C07282=1047.858,-113.181,431.059,169.619,31.732,156.022
C07283=1047.864,-112.931,431.049,169.621,31.732,156.022
C07284=1047.869,-112.682,431.040,169.623,31.732,156.022
C07285=1047.875,-112.432,431.030,169.626,31.733,156.022
C07286=1047.881,-112.182,431.020,169.628,31.733,156.022
C07287=1047.887,-111.932,431.011,169.630,31.733,156.022
C07288=1047.894,-111.683,431.000,169.632,31.733,156.021
C07289=1047.900,-111.433,430.991,169.635,31.734,156.022
C07290=1047.906,-111.183,430.981,169.637,31.735,156.021
C07291=1047.912,-110.933,430.972,169.639,31.735,156.021
C07292=1047.918,-110.684,430.962,169.642,31.735,156.021
C07293=1047.924,-110.434,430.953,169.644,31.736,156.021
C07294=1047.931,-110.184,430.943,169.646,31.736,156.021
C07295=1047.937,-109.935,430.933,169.648,31.736,156.021
C07296=1047.942,-109.685,430.923,169.650,31.736,156.021
C07297=1047.949,-109.435,430.913,169.652,31.737,156.021
C07298=1047.955,-109.185,430.903,169.654,31.737,156.021
C07299=1047.961,-108.935,430.894,169.656,31.738,156.021
C07300=1047.967,-108.686,430.884,169.659,31.738,156.021
C07301=1047.974,-108.436,430.874,169.661,31.738,156.021
C07302=1047.980,-108.187,430.864,169.663,31.739,156.021
C07303=1047.986,-107.937,430.855,169.666,31.739,156.021
C07304=1047.992,-107.687,430.845,169.668,31.739,156.021
C07305=1047.998,-107.437,430.834,169.670,31.740,156.021
C07306=1048.005,-107.187,430.825,169.672,31.741,156.021
C07307=1048.011,-106.937,430.815,169.675,31.741,156.021
C07308=1048.017,-106.687,430.805,169.677,31.741,156.021
C07309=1048.023,-106.438,430.795,169.679,31.741,156.020
C07310=1048.029,-106.188,430.785,169.681,31.742,156.021
C07311=1048.035,-105.938,430.775,169.684,31.743,156.020
C07312=1048.042,-105.689,430.765,169.686,31.743,156.020
C07313=1048.047,-105.439,430.755,169.687,31.743,156.020
C07314=1048.053,-105.189,430.745,169.690,31.744,156.020
C07315=1048.060,-104.940,430.735,169.692,31.745,156.020
C07316=1048.066,-104.690,430.726,169.694,31.745,156.020
C07317=1048.071,-104.440,430.715,169.696,31.746,156.020
C07318=1048.078,-104.191,430.705,169.699,31.746,156.020
C07319=1048.084,-103.941,430.696,169.701,31.746,156.020
C07320=1048.090,-103.691,430.686,169.703,31.747,156.020
C07321=1048.096,-103.441,430.675,169.705,31.747,156.020
C07322=1048.103,-103.191,430.665,169.708,31.748,156.020
C07323=1048.109,-102.942,430.655,169.710,31.749,156.020
C07324=1048.114,-102.692,430.645,169.712,31.749,156.020
C07325=1048.121,-102.442,430.635,169.714,31.749,156.020
C07326=1048.127,-102.193,430.625,169.717,31.750,156.020
C07327=1048.133,-101.943,430.615,169.719,31.751,156.020
C07328=1048.139,-101.694,430.604,169.721,31.751,156.020
C07329=1048.145,-101.444,430.595,169.723,31.752,156.020
C07330=1048.152,-101.194,430.584,169.725,31.752,156.020
C07331=1048.158,-100.944,430.574,169.727,31.752,156.020
C07332=1048.164,-100.695,430.564,169.729,31.753,156.020
C07333=1048.170,-100.445,430.554,169.731,31.753,156.020
C07334=1048.176,-100.196,430.543,169.734,31.754,156.020
C07335=1048.182,-99.946,430.534,169.736,31.755,156.020
C07336=1048.189,-99.659,430.521,169.739,31.756,156.020
C07337=1048.196,-99.373,430.510,169.741,31.756,156.020
C07338=1048.203,-99.085,430.498,169.744,31.756,156.020
C07339=1048.211,-98.799,430.486,169.746,31.757,156.020
C07340=1048.220,-98.428,430.471,169.750,31.758,156.020
C07341=1048.229,-98.056,430.456,169.753,31.759,156.020
C07342=1048.238,-97.685,430.441,169.756,31.760,156.020
C07343=1048.247,-97.313,430.425,169.760,31.761,156.020
C07344=1048.254,-97.063,430.415,169.761,31.761,156.020
C07345=1048.259,-96.814,430.404,169.763,31.762,156.020
C07346=1048.266,-96.564,430.394,169.765,31.762,156.020
C07347=1048.272,-96.314,430.383,169.768,31.763,156.020
C07348=1048.278,-96.064,430.373,169.770,31.764,156.020
C07349=1048.284,-95.815,430.362,169.772,31.764,156.020
C07350=1048.290,-95.565,430.352,169.774,31.765,156.020
C07351=1048.296,-95.316,430.342,169.776,31.766,156.020
C07352=1048.302,-95.065,430.331,169.779,31.767,156.020
C07353=1048.309,-94.816,430.321,169.781,31.768,156.020
C07354=1048.314,-94.566,430.310,169.783,31.768,156.020
C07355=1048.320,-94.317,430.299,169.785,31.769,156.020
C07356=1048.326,-94.067,430.290,169.788,31.770,156.020
C07357=1048.333,-93.817,430.278,169.790,31.770,156.020
C07358=1048.339,-93.568,430.268,169.792,31.771,156.020
C07359=1048.345,-93.318,430.257,169.793,31.772,156.020
C07360=1048.350,-93.068,430.247,169.795,31.772,156.020
C07361=1048.357,-92.818,430.236,169.798,31.773,156.020
C07362=1048.363,-92.569,430.226,169.800,31.774,156.020
C07363=1048.369,-92.319,430.215,169.802,31.774,156.020
C07364=1048.375,-92.070,430.204,169.804,31.775,156.020
C07365=1048.381,-91.819,430.194,169.806,31.776,156.020
C07366=1048.388,-91.570,430.184,169.809,31.777,156.020
C07367=1048.393,-91.320,430.173,169.811,31.777,156.020
C07368=1048.400,-91.070,430.161,169.813,31.778,156.020
C07369=1048.406,-90.821,430.151,169.815,31.779,156.020
C07370=1048.412,-90.571,430.141,169.818,31.779,156.020
C07371=1048.418,-90.321,430.130,169.820,31.780,156.020
C07372=1048.425,-90.072,430.120,169.822,31.781,156.020
C07373=1048.430,-89.822,430.109,169.824,31.782,156.020
C07374=1048.437,-89.572,430.098,169.826,31.782,156.020
C07375=1048.443,-89.323,430.087,169.828,31.783,156.020
C07376=1048.449,-89.073,430.076,169.830,31.784,156.020
C07377=1048.456,-88.823,430.066,169.832,31.785,156.020
C07378=1048.461,-88.573,430.055,169.834,31.785,156.020
C07379=1048.467,-88.324,430.045,169.836,31.786,156.020
C07380=1048.474,-88.074,430.034,169.839,31.787,156.020
C07381=1048.480,-87.824,430.023,169.841,31.788,156.020
C07382=1048.486,-87.575,430.012,169.843,31.788,156.020
C07383=1048.493,-87.325,430.001,169.845,31.789,156.020
C07384=1048.498,-87.075,429.991,169.847,31.790,156.020
C07385=1048.504,-86.826,429.980,169.850,31.791,156.020
C07386=1048.511,-86.576,429.969,169.852,31.791,156.020
C07387=1048.517,-86.327,429.958,169.854,31.792,156.020
C07388=1048.523,-86.076,429.947,169.856,31.793,156.020
C07389=1048.530,-85.827,429.937,169.858,31.794,156.020
C07390=1048.536,-85.578,429.926,169.860,31.795,156.021
C07391=1048.542,-85.328,429.915,169.862,31.795,156.020
C07392=1048.548,-85.078,429.904,169.864,31.796,156.021
C07393=1048.555,-84.828,429.893,169.866,31.797,156.021
C07394=1048.560,-84.579,429.882,169.869,31.798,156.021
C07395=1048.567,-84.329,429.871,169.871,31.799,156.021
C07396=1048.577,-83.916,429.853,169.874,31.800,156.021
C07397=1048.588,-83.505,429.835,169.878,31.801,156.021
C07398=1048.598,-83.092,429.818,169.882,31.803,156.021
C07399=1048.608,-82.680,429.799,169.885,31.804,156.021
C07400=1048.615,-82.431,429.788,169.887,31.805,156.021
C07401=1048.621,-82.181,429.777,169.890,31.806,156.021
C07402=1048.627,-81.931,429.766,169.891,31.807,156.021
C07403=1048.633,-81.682,429.756,169.893,31.807,156.021
C07404=1048.640,-81.431,429.745,169.895,31.808,156.021
C07405=1048.645,-81.182,429.734,169.897,31.809,156.021
C07406=1048.652,-80.932,429.722,169.900,31.810,156.021
C07407=1048.659,-80.683,429.711,169.902,31.810,156.021
C07408=1048.665,-80.433,429.700,169.904,31.811,156.021
C07409=1048.671,-80.184,429.689,169.906,31.812,156.021
C07410=1048.677,-79.933,429.678,169.908,31.813,156.021
C07411=1048.683,-79.684,429.668,169.911,31.814,156.021
C07412=1048.690,-79.435,429.656,169.913,31.815,156.021
C07413=1048.696,-79.185,429.645,169.915,31.816,156.021
C07414=1048.702,-78.935,429.634,169.917,31.817,156.022
C07415=1048.708,-78.685,429.623,169.919,31.818,156.022
C07416=1048.715,-78.436,429.611,169.921,31.819,156.022
C07417=1048.720,-78.186,429.600,169.923,31.820,156.022
C07418=1048.727,-77.936,429.589,169.925,31.820,156.022
C07419=1048.732,-77.687,429.578,169.927,31.821,156.022
C07420=1048.739,-77.437,429.566,169.929,31.822,156.022
C07421=1048.745,-77.188,429.555,169.931,31.823,156.022
C07422=1048.751,-76.937,429.544,169.933,31.825,156.022
C07423=1048.757,-76.689,429.532,169.935,31.825,156.022
C07424=1048.764,-76.438,429.521,169.938,31.826,156.022
C07425=1048.770,-76.188,429.510,169.940,31.827,156.022
C07426=1048.776,-75.939,429.498,169.942,31.828,156.022
C07427=1048.782,-75.689,429.487,169.944,31.829,156.022
C07428=1048.788,-75.440,429.476,169.946,31.830,156.022
C07429=1048.795,-75.190,429.464,169.948,31.831,156.022
C07430=1048.800,-74.941,429.453,169.951,31.832,156.022
C07431=1048.807,-74.690,429.442,169.952,31.833,156.023
C07432=1048.813,-74.441,429.430,169.954,31.834,156.023
C07433=1048.819,-74.191,429.419,169.956,31.835,156.023
C07434=1048.826,-73.942,429.407,169.958,31.836,156.023
C07435=1048.831,-73.692,429.396,169.960,31.837,156.023
C07436=1048.838,-73.443,429.384,169.962,31.838,156.023
C07437=1048.844,-73.193,429.373,169.965,31.839,156.023
C07438=1048.849,-72.943,429.362,169.967,31.840,156.023
C07439=1048.856,-72.694,429.350,169.969,31.841,156.023
C07440=1048.862,-72.444,429.339,169.971,31.843,156.023
C07441=1048.868,-72.194,429.327,169.973,31.843,156.023
C07442=1048.874,-71.945,429.316,169.975,31.844,156.023
C07443=1048.880,-71.695,429.303,169.977,31.846,156.024
C07444=1048.886,-71.445,429.292,169.979,31.847,156.024
C07445=1048.893,-71.196,429.280,169.981,31.848,156.024
C07446=1048.898,-70.946,429.270,169.983,31.849,156.024
C07447=1048.904,-70.696,429.257,169.985,31.850,156.024
C07448=1048.911,-70.447,429.245,169.987,31.851,156.024
C07449=1048.917,-70.197,429.234,169.989,31.853,156.024
C07450=1048.923,-69.948,429.222,169.991,31.853,156.024
C07451=1048.929,-69.697,429.210,169.993,31.854,156.024
C07452=1048.935,-69.448,429.199,169.996,31.856,156.024
C07453=1048.941,-69.198,429.188,169.998,31.857,156.025
C07454=1048.947,-68.949,429.176,170.000,31.858,156.025
C07455=1048.953,-68.699,429.163,170.002,31.859,156.025
C07456=1048.959,-68.449,429.152,170.004,31.860,156.025
C07457=1048.966,-68.200,429.141,170.006,31.861,156.025
C07458=1048.971,-67.950,429.129,170.007,31.862,156.025
C07459=1048.978,-67.700,429.117,170.009,31.863,156.025
C07460=1048.984,-67.419,429.103,170.012,31.865,156.025
C07461=1048.991,-67.136,429.090,170.014,31.866,156.025
C07462=1048.999,-66.854,429.077,170.017,31.867,156.025
C07463=1049.006,-66.572,429.064,170.019,31.868,156.025
C07464=1049.011,-66.322,429.052,170.021,31.870,156.026
C07465=1049.017,-66.073,429.040,170.023,31.871,156.026
C07466=1049.024,-65.823,429.028,170.025,31.872,156.026
C07467=1049.030,-65.573,429.017,170.027,31.873,156.026
C07468=1049.036,-65.323,429.004,170.029,31.874,156.026
C07469=1049.042,-65.074,428.993,170.032,31.876,156.026
C07470=1049.049,-64.824,428.982,170.034,31.876,156.026
C07471=1049.055,-64.574,428.969,170.035,31.878,156.026
C07472=1049.061,-64.326,428.957,170.037,31.879,156.026
C07473=1049.067,-64.076,428.946,170.039,31.880,156.027
C07474=1049.073,-63.825,428.934,170.041,31.881,156.027
C07475=1049.080,-63.576,428.922,170.043,31.882,156.027
C07476=1049.086,-63.327,428.910,170.045,31.884,156.027
C07477=1049.092,-63.077,428.898,170.047,31.884,156.027
C07478=1049.098,-62.828,428.886,170.050,31.886,156.027
C07479=1049.105,-62.577,428.874,170.052,31.887,156.027
C07480=1049.110,-62.327,428.862,170.054,31.888,156.027
C07481=1049.116,-62.079,428.850,170.056,31.889,156.027
C07482=1049.123,-61.829,428.838,170.058,31.890,156.027
C07483=1049.129,-61.579,428.826,170.060,31.892,156.028
C07484=1049.135,-61.329,428.814,170.062,31.892,156.028
C07485=1049.141,-61.080,428.803,170.063,31.894,156.028
C07486=1049.147,-60.830,428.790,170.065,31.895,156.028
C07487=1049.154,-60.581,428.778,170.067,31.896,156.028
C07488=1049.161,-60.331,428.766,170.069,31.897,156.028
C07489=1049.167,-60.081,428.754,170.072,31.899,156.028
C07490=1049.173,-59.832,428.742,170.074,31.900,156.028
C07491=1049.179,-59.583,428.730,170.076,31.901,156.028
C07492=1049.185,-59.333,428.718,170.078,31.902,156.029
C07493=1049.191,-59.083,428.706,170.080,31.904,156.029
C07494=1049.198,-58.833,428.695,170.082,31.904,156.029
C07495=1049.204,-58.583,428.682,170.084,31.906,156.029
C07496=1049.211,-58.334,428.670,170.086,31.907,156.029
C07497=1049.217,-58.084,428.658,170.088,31.908,156.029
C07498=1049.223,-57.835,428.646,170.090,31.909,156.029
C07499=1049.229,-57.585,428.634,170.091,31.911,156.029
C07500=1049.235,-57.335,428.621,170.094,31.912,156.029
C07501=1049.242,-57.086,428.609,170.096,31.913,156.030
C07502=1049.248,-56.836,428.597,170.098,31.914,156.030
C07503=1049.254,-56.586,428.585,170.100,31.916,156.030
C07504=1049.261,-56.337,428.573,170.102,31.916,156.030
C07505=1049.268,-56.087,428.561,170.104,31.918,156.030
C07506=1049.274,-55.837,428.548,170.106,31.919,156.030
C07507=1049.280,-55.589,428.537,170.108,31.920,156.030
C07508=1049.286,-55.339,428.524,170.110,31.922,156.030
C07509=1049.292,-55.089,428.512,170.112,31.923,156.031
C07510=1049.299,-54.839,428.500,170.114,31.924,156.031
C07511=1049.305,-54.590,428.488,170.116,31.925,156.031
C07512=1049.311,-54.340,428.476,170.118,31.927,156.031
C07513=1049.317,-54.090,428.463,170.120,31.927,156.031
C07514=1049.324,-53.841,428.451,170.122,31.929,156.031
C07515=1049.331,-53.592,428.439,170.124,31.930,156.031
C07516=1049.337,-53.342,428.426,170.126,31.931,156.031
C07517=1049.343,-53.092,428.414,170.128,31.933,156.032
C07518=1049.349,-52.842,428.402,170.130,31.934,156.032
C07519=1049.356,-52.593,428.390,170.132,31.935,156.032
C07520=1049.362,-52.343,428.377,170.134,31.936,156.032
C07521=1049.369,-52.093,428.365,170.136,31.938,156.032
C07522=1049.375,-51.844,428.353,170.138,31.938,156.032
C07523=1049.381,-51.594,428.340,170.140,31.940,156.032
C07524=1049.389,-51.313,428.327,170.143,31.942,156.032
C07525=1049.395,-51.033,428.313,170.145,31.943,156.033
C07526=1049.403,-50.751,428.299,170.146,31.944,156.033
C07527=1049.410,-50.471,428.285,170.149,31.946,156.033
C07528=1049.416,-50.222,428.272,170.151,31.947,156.033
C07529=1049.422,-49.972,428.259,170.153,31.949,156.033
C07530=1049.429,-49.722,428.247,170.155,31.950,156.033
C07531=1049.435,-49.472,428.235,170.157,31.951,156.033
C07532=1049.441,-49.222,428.222,170.159,31.952,156.034
C07533=1049.447,-48.973,428.209,170.161,31.954,156.034
C07534=1049.454,-48.724,428.197,170.163,31.955,156.034
C07535=1049.460,-48.474,428.184,170.165,31.957,156.034
C07536=1049.466,-48.224,428.171,170.167,31.958,156.034
C07537=1049.472,-47.975,428.159,170.169,31.959,156.034
C07538=1049.478,-47.725,428.147,170.171,31.961,156.034
C07539=1049.485,-47.476,428.133,170.172,31.962,156.035
C07540=1049.490,-47.226,428.121,170.174,31.964,156.035
C07541=1049.496,-46.976,428.108,170.176,31.965,156.035
C07542=1049.503,-46.727,428.095,170.178,31.966,156.035
C07543=1049.509,-46.477,428.083,170.180,31.967,156.035
C07544=1049.515,-46.227,428.071,170.182,31.969,156.035
C07545=1049.521,-45.978,428.057,170.184,31.970,156.036
C07546=1049.527,-45.728,428.045,170.186,31.972,156.036
C07547=1049.534,-45.479,428.032,170.188,31.973,156.036
C07548=1049.540,-45.229,428.020,170.190,31.975,156.036
C07549=1049.546,-44.979,428.007,170.192,31.976,156.036
C07550=1049.552,-44.730,427.994,170.194,31.977,156.036
C07551=1049.558,-44.480,427.981,170.196,31.979,156.036
C07552=1049.565,-44.231,427.968,170.197,31.980,156.037
C07553=1049.571,-43.981,427.956,170.199,31.982,156.037
C07554=1049.577,-43.731,427.943,170.201,31.983,156.037
C07555=1049.583,-43.482,427.930,170.203,31.985,156.037
C07556=1049.590,-43.232,427.917,170.205,31.986,156.037
C07557=1049.597,-42.983,427.904,170.207,31.987,156.037
C07558=1049.603,-42.733,427.892,170.209,31.989,156.038
C07559=1049.609,-42.484,427.879,170.211,31.990,156.038
C07560=1049.615,-42.234,427.866,170.213,31.992,156.038
C07561=1049.621,-41.984,427.853,170.215,31.993,156.038
C07562=1049.627,-41.735,427.841,170.217,31.995,156.038
C07563=1049.634,-41.486,427.828,170.219,31.996,156.038
C07564=1049.640,-41.236,427.815,170.221,31.997,156.039
C07565=1049.646,-40.986,427.801,170.223,31.999,156.039
C07566=1049.652,-40.736,427.789,170.224,32.000,156.039
C07567=1049.659,-40.487,427.776,170.226,32.001,156.039
C07568=1049.666,-40.238,427.763,170.228,32.003,156.039
C07569=1049.671,-39.988,427.750,170.230,32.004,156.039
C07570=1049.678,-39.738,427.737,170.232,32.006,156.040
C07571=1049.684,-39.489,427.725,170.234,32.007,156.040
C07572=1049.690,-39.239,427.711,170.236,32.009,156.040
C07573=1049.697,-38.990,427.698,170.238,32.010,156.040
C07574=1049.703,-38.740,427.686,170.240,32.012,156.040
C07575=1049.709,-38.490,427.672,170.242,32.013,156.040
C07576=1049.715,-38.241,427.660,170.244,32.015,156.041
C07577=1049.722,-37.991,427.647,170.246,32.016,156.041
C07578=1049.728,-37.742,427.633,170.248,32.018,156.041
C07579=1049.734,-37.491,427.620,170.249,32.019,156.041
C07580=1049.740,-37.242,427.607,170.251,32.021,156.041
C07581=1049.746,-36.993,427.593,170.253,32.022,156.041
C07582=1049.752,-36.743,427.581,170.255,32.024,156.042
C07583=1049.758,-36.494,427.567,170.257,32.025,156.042
C07584=1049.764,-36.244,427.554,170.259,32.027,156.042
C07585=1049.771,-35.994,427.541,170.261,32.028,156.042
C07586=1049.777,-35.744,427.528,170.263,32.030,156.042
C07587=1049.783,-35.495,427.515,170.265,32.032,156.043
C07588=1049.790,-35.215,427.500,170.267,32.033,156.043
C07589=1049.797,-34.935,427.485,170.269,32.035,156.043
C07590=1049.804,-34.655,427.470,170.272,32.037,156.043
C07591=1049.811,-34.373,427.455,170.274,32.038,156.043
C07592=1049.817,-34.124,427.442,170.275,32.040,156.044
C07593=1049.823,-33.875,427.429,170.277,32.041,156.044
C07594=1049.830,-33.625,427.416,170.279,32.043,156.044
C07595=1049.837,-33.375,427.402,170.281,32.044,156.044
C07596=1049.842,-33.126,427.389,170.283,32.046,156.044
C07597=1049.849,-32.876,427.376,170.285,32.048,156.045
C07598=1049.855,-32.627,427.363,170.286,32.049,156.045
C07599=1049.861,-32.378,427.350,170.288,32.051,156.045
C07600=1049.867,-32.127,427.335,170.290,32.052,156.045
C07601=1049.873,-31.878,427.322,170.292,32.054,156.045
C07602=1049.879,-31.628,427.309,170.294,32.055,156.045
C07603=1049.886,-31.378,427.296,170.296,32.057,156.046
C07604=1049.892,-31.129,427.283,170.298,32.058,156.046
C07605=1049.899,-30.880,427.269,170.300,32.060,156.046
C07606=1049.905,-30.631,427.256,170.301,32.062,156.046
C07607=1049.912,-30.381,427.242,170.303,32.063,156.046
C07608=1049.918,-30.131,427.229,170.305,32.065,156.047
C07609=1049.923,-29.882,427.215,170.307,32.066,156.047
C07610=1049.930,-29.632,427.202,170.309,32.068,156.047
C07611=1049.936,-29.383,427.188,170.311,32.069,156.047
C07612=1049.942,-29.133,427.175,170.313,32.070,156.047
C07613=1049.948,-28.883,427.163,170.315,32.073,156.048
C07614=1049.955,-28.633,427.149,170.317,32.074,156.048
C07615=1049.961,-28.384,427.136,170.319,32.076,156.048
C07616=1049.968,-28.135,427.122,170.321,32.077,156.048
C07617=1049.974,-27.885,427.108,170.323,32.078,156.048
C07618=1049.980,-27.635,427.095,170.324,32.080,156.048
C07619=1049.987,-27.385,427.081,170.326,32.081,156.049
C07620=1049.993,-27.136,427.068,170.327,32.083,156.049
C07621=1049.999,-26.887,427.055,170.329,32.085,156.049
C07622=1050.006,-26.637,427.041,170.331,32.086,156.049
C07623=1050.011,-26.387,427.027,170.333,32.088,156.049
C07624=1050.018,-26.138,427.014,170.335,32.090,156.050
C07625=1050.024,-25.888,426.999,170.337,32.091,156.050
C07626=1050.030,-25.639,426.986,170.339,32.093,156.050
C07627=1050.036,-25.390,426.972,170.341,32.095,156.050
C07628=1050.043,-25.140,426.958,170.343,32.096,156.051
C07629=1050.049,-24.890,426.945,170.345,32.098,156.051
C07630=1050.055,-24.641,426.932,170.347,32.099,156.051
C07631=1050.061,-24.391,426.917,170.348,32.101,156.051
C07632=1050.067,-24.142,426.904,170.350,32.103,156.051
C07633=1050.073,-23.892,426.891,170.352,32.104,156.052
C07634=1050.080,-23.643,426.876,170.353,32.106,156.052
C07635=1050.086,-23.393,426.863,170.355,32.108,156.052
C07636=1050.092,-23.144,426.849,170.357,32.109,156.052
C07637=1050.098,-22.894,426.835,170.359,32.111,156.052
C07638=1050.105,-22.645,426.822,170.361,32.113,156.053
C07639=1050.111,-22.394,426.808,170.363,32.114,156.053
C07640=1050.117,-22.146,426.794,170.365,32.117,156.053
C07641=1050.123,-21.896,426.780,170.366,32.118,156.053
C07642=1050.129,-21.646,426.766,170.368,32.119,156.054
C07643=1050.136,-21.397,426.753,170.370,32.121,156.054
C07644=1050.142,-21.147,426.739,170.372,32.123,156.054
C07645=1050.148,-20.898,426.725,170.374,32.124,156.054
C07646=1050.154,-20.648,426.711,170.376,32.126,156.054
C07647=1050.161,-20.398,426.697,170.377,32.128,156.055
C07648=1050.167,-20.149,426.684,170.379,32.129,156.055
C07649=1050.173,-19.899,426.669,170.381,32.131,156.055
C07650=1050.179,-19.650,426.656,170.383,32.133,156.055
C07651=1050.185,-19.400,426.641,170.384,32.134,156.055
C07652=1050.193,-19.119,426.626,170.387,32.137,156.056
C07653=1050.200,-18.838,426.611,170.389,32.138,156.056
C07654=1050.207,-18.557,426.595,170.391,32.140,156.056
C07655=1050.214,-18.276,426.579,170.393,32.142,156.056
C07656=1050.219,-18.026,426.565,170.395,32.144,156.057
C07657=1050.227,-17.777,426.551,170.397,32.145,156.057
C07658=1050.233,-17.528,426.538,170.399,32.147,156.057
C07659=1050.239,-17.277,426.523,170.401,32.149,156.057
C07660=1050.245,-17.029,426.509,170.402,32.150,156.058
C07661=1050.251,-16.778,426.495,170.403,32.152,156.058
C07662=1050.258,-16.529,426.482,170.405,32.154,156.058
C07663=1050.264,-16.279,426.467,170.407,32.155,156.058
C07664=1050.270,-16.030,426.454,170.409,32.157,156.058
C07665=1050.277,-15.781,426.439,170.411,32.159,156.059
C07666=1050.283,-15.531,426.425,170.413,32.161,156.059
C07667=1050.290,-15.281,426.412,170.415,32.162,156.059
C07668=1050.296,-15.032,426.397,170.416,32.164,156.059
C07669=1050.301,-14.782,426.383,170.418,32.166,156.060
C07670=1050.309,-14.533,426.369,170.420,32.167,156.060
C07671=1050.314,-14.283,426.355,170.422,32.169,156.060
C07672=1050.320,-14.033,426.340,170.424,32.171,156.060
C07673=1050.327,-13.784,426.327,170.426,32.173,156.061
C07674=1050.333,-13.535,426.312,170.428,32.174,156.061
C07675=1050.339,-13.285,426.298,170.429,32.176,156.061
C07676=1050.346,-13.036,426.283,170.430,32.178,156.061
C07677=1050.351,-12.786,426.270,170.432,32.180,156.061
C07678=1050.358,-12.536,426.255,170.434,32.181,156.062
C07679=1050.364,-12.287,426.241,170.436,32.183,156.062
C07680=1050.370,-12.037,426.226,170.438,32.185,156.062
C07681=1050.376,-11.788,426.213,170.440,32.187,156.062
C07682=1050.383,-11.539,426.198,170.441,32.188,156.063
C07683=1050.388,-11.289,426.184,170.443,32.190,156.063
C07684=1050.395,-11.039,426.169,170.445,32.192,156.063
C07685=1050.401,-10.789,426.156,170.447,32.194,156.063
C07686=1050.407,-10.540,426.141,170.449,32.195,156.064
C07687=1050.414,-10.291,426.126,170.451,32.197,156.064
C07688=1050.420,-10.041,426.113,170.453,32.199,156.064
C07689=1050.426,-9.792,426.098,170.454,32.201,156.064
C07690=1050.432,-9.542,426.084,170.456,32.202,156.064
C07691=1050.438,-9.293,426.069,170.457,32.204,156.065
C07692=1050.445,-9.043,426.055,170.459,32.206,156.065
C07693=1050.451,-8.794,426.041,170.461,32.208,156.065
C07694=1050.457,-8.544,426.026,170.463,32.209,156.065
C07695=1050.464,-8.295,426.012,170.464,32.211,156.066
C07696=1050.470,-8.045,425.998,170.466,32.213,156.066
C07697=1050.476,-7.795,425.983,170.468,32.215,156.066
C07698=1050.482,-7.547,425.969,170.470,32.217,156.067
C07699=1050.489,-7.297,425.955,170.472,32.218,156.067
C07700=1050.495,-7.047,425.940,170.474,32.221,156.067
C07701=1050.501,-6.798,425.925,170.475,32.222,156.067
C07702=1050.508,-6.548,425.912,170.477,32.224,156.067
C07703=1050.513,-6.299,425.897,170.479,32.225,156.068
C07704=1050.520,-6.049,425.882,170.481,32.228,156.068
C07705=1050.526,-5.800,425.867,170.482,32.229,156.068
C07706=1050.532,-5.550,425.854,170.484,32.231,156.068
C07707=1050.539,-5.301,425.839,170.485,32.232,156.069
C07708=1050.545,-5.051,425.824,170.487,32.235,156.069
C07709=1050.551,-4.802,425.809,170.489,32.236,156.069
C07710=1050.558,-4.552,425.796,170.491,32.238,156.069
C07711=1050.564,-4.303,425.781,170.493,32.240,156.070
C07712=1050.570,-4.053,425.766,170.495,32.242,156.070
C07713=1050.577,-3.804,425.752,170.496,32.243,156.070
C07714=1050.583,-3.554,425.738,170.498,32.245,156.070
C07715=1050.589,-3.304,425.723,170.500,32.247,156.071
C07716=1050.596,-3.022,425.706,170.502,32.249,156.071
C07717=1050.604,-2.739,425.689,170.504,32.251,156.071
C07718=1050.610,-2.457,425.673,170.506,32.253,156.072
C07719=1050.617,-2.174,425.656,170.508,32.255,156.072
C07720=1050.622,-1.924,425.641,170.509,32.257,156.072
C07721=1050.629,-1.675,425.626,170.511,32.259,156.072
C07722=1050.635,-1.425,425.611,170.513,32.261,156.073
C07723=1050.641,-1.176,425.597,170.514,32.263,156.073
C07724=1050.647,-0.926,425.582,170.516,32.265,156.073
C07725=1050.654,-0.676,425.567,170.518,32.267,156.073
C07726=1050.659,-0.427,425.552,170.520,32.269,156.074
C07727=1050.666,-0.178,425.537,170.522,32.271,156.074
C07728=1050.672,0.072,425.523,170.523,32.272,156.074
C07729=1050.678,0.321,425.508,170.525,32.274,156.074
C07730=1050.684,0.571,425.493,170.527,32.276,156.075
C07731=1050.691,0.820,425.478,170.529,32.278,156.075
C07732=1050.697,1.070,425.463,170.531,32.280,156.075
C07733=1050.703,1.319,425.449,170.532,32.282,156.076
C07734=1050.709,1.569,425.434,170.534,32.284,156.076
C07735=1050.716,1.818,425.419,170.536,32.285,156.076
C07736=1050.722,2.068,425.404,170.537,32.287,156.076
C07737=1050.728,2.317,425.389,170.538,32.289,156.077
C07738=1050.734,2.567,425.374,170.540,32.291,156.077
C07739=1050.740,2.816,425.359,170.542,32.293,156.077
C07740=1050.746,3.065,425.344,170.544,32.295,156.077
C07741=1050.752,3.315,425.329,170.546,32.297,156.078
C07742=1050.758,3.565,425.314,170.547,32.299,156.078
C07743=1050.765,3.814,425.299,170.549,32.300,156.078
C07744=1050.771,4.064,425.284,170.551,32.302,156.078
C07745=1050.777,4.313,425.270,170.553,32.305,156.079
C07746=1050.784,4.562,425.254,170.554,32.306,156.079
C07747=1050.790,4.812,425.239,170.556,32.308,156.079
C07748=1050.796,5.061,425.224,170.558,32.310,156.080
C07749=1050.802,5.310,425.210,170.560,32.312,156.080
C07750=1050.808,5.560,425.195,170.562,32.314,156.080
C07751=1050.814,5.810,425.179,170.563,32.315,156.080
C07752=1050.820,6.060,425.164,170.564,32.318,156.081
C07753=1050.827,6.309,425.149,170.566,32.320,156.081
C07754=1050.834,6.558,425.133,170.568,32.321,156.081
C07755=1050.839,6.807,425.119,170.569,32.323,156.081
C07756=1050.846,7.057,425.104,170.571,32.325,156.082
C07757=1050.852,7.307,425.089,170.573,32.327,156.082
C07758=1050.858,7.556,425.074,170.575,32.329,156.082
C07759=1050.865,7.806,425.059,170.577,32.331,156.082
C07760=1050.871,8.055,425.043,170.578,32.333,156.083
C07761=1050.877,8.304,425.028,170.580,32.334,156.083
C07762=1050.883,8.554,425.013,170.582,32.336,156.083
C07763=1050.889,8.804,424.998,170.584,32.338,156.084
C07764=1050.896,9.053,424.983,170.585,32.340,156.084
C07765=1050.902,9.302,424.968,170.587,32.342,156.084
C07766=1050.909,9.552,424.953,170.589,32.344,156.084
C07767=1050.915,9.802,424.938,170.591,32.346,156.085
C07768=1050.921,10.051,424.922,170.592,32.348,156.085
C07769=1050.927,10.300,424.907,170.593,32.349,156.085
C07770=1050.933,10.549,424.892,170.595,32.351,156.085
C07771=1050.940,10.799,424.877,170.597,32.353,156.086
C07772=1050.946,11.048,424.862,170.599,32.355,156.086
C07773=1050.953,11.298,424.847,170.600,32.357,156.086
C07774=1050.959,11.547,424.832,170.602,32.359,156.087
C07775=1050.965,11.797,424.816,170.604,32.361,156.087
C07776=1050.971,12.046,424.800,170.606,32.362,156.087
C07777=1050.978,12.296,424.785,170.607,32.364,156.087
C07778=1050.984,12.546,424.771,170.609,32.366,156.088
C07779=1050.991,12.795,424.755,170.611,32.368,156.088
C07780=1050.998,13.079,424.738,170.613,32.371,156.088
C07781=1051.005,13.364,424.720,170.615,32.373,156.088
C07782=1051.012,13.649,424.703,170.617,32.375,156.089
C07783=1051.019,13.934,424.685,170.619,32.377,156.089
C07784=1051.026,14.183,424.670,170.621,32.379,156.089
C07785=1051.032,14.432,424.655,170.622,32.381,156.090
C07786=1051.038,14.682,424.639,170.623,32.383,156.090
C07787=1051.045,14.931,424.623,170.625,32.384,156.090
C07788=1051.051,15.181,424.608,170.627,32.386,156.090
C07789=1051.057,15.430,424.592,170.628,32.388,156.091
C07790=1051.063,15.680,424.577,170.630,32.390,156.091
C07791=1051.069,15.929,424.561,170.632,32.392,156.091
C07792=1051.076,16.179,424.546,170.634,32.394,156.092
C07793=1051.082,16.428,424.530,170.635,32.396,156.092
C07794=1051.087,16.677,424.515,170.637,32.398,156.092
C07795=1051.094,16.926,424.500,170.639,32.400,156.092
C07796=1051.100,17.176,424.484,170.640,32.402,156.093
C07797=1051.107,17.425,424.468,170.642,32.404,156.093
C07798=1051.113,17.675,424.453,170.644,32.406,156.093
C07799=1051.119,17.924,424.437,170.646,32.408,156.094
C07800=1051.125,18.174,424.422,170.647,32.410,156.094
C07801=1051.131,18.423,424.406,170.649,32.412,156.094
C07802=1051.138,18.673,424.391,170.651,32.414,156.094
C07803=1051.144,18.922,424.375,170.652,32.416,156.095
C07804=1051.150,19.172,424.360,170.653,32.418,156.095
C07805=1051.157,19.421,424.344,170.655,32.420,156.095
C07806=1051.163,19.670,424.328,170.657,32.422,156.096
C07807=1051.169,19.920,424.313,170.658,32.424,156.096
C07808=1051.175,20.169,424.297,170.660,32.426,156.096
C07809=1051.181,20.419,424.282,170.662,32.428,156.097
C07810=1051.187,20.668,424.265,170.664,32.430,156.097
C07811=1051.194,20.917,424.250,170.665,32.431,156.097
C07812=1051.200,21.167,424.234,170.667,32.433,156.097
C07813=1051.206,21.416,424.219,170.669,32.435,156.098
C07814=1051.212,21.666,424.202,170.671,32.437,156.098
C07815=1051.219,21.915,424.187,170.672,32.439,156.098
C07816=1051.225,22.165,424.171,170.674,32.441,156.099
C07817=1051.231,22.414,424.156,170.676,32.443,156.099
C07818=1051.237,22.664,424.140,170.677,32.445,156.099
C07819=1051.243,22.913,424.124,170.679,32.447,156.099
C07820=1051.250,23.163,424.108,170.681,32.449,156.100
C07821=1051.256,23.413,424.092,170.682,32.451,156.100
C07822=1051.262,23.662,424.076,170.683,32.453,156.100
C07823=1051.268,23.911,424.060,170.685,32.456,156.101
C07824=1051.275,24.160,424.045,170.687,32.458,156.101
C07825=1051.281,24.410,424.029,170.688,32.460,156.101
C07826=1051.287,24.660,424.013,170.690,32.461,156.101
C07827=1051.293,24.909,423.997,170.692,32.463,156.102
C07828=1051.299,25.158,423.981,170.693,32.465,156.102
C07829=1051.306,25.408,423.966,170.695,32.467,156.102
C07830=1051.312,25.657,423.950,170.697,32.469,156.103
C07831=1051.318,25.906,423.934,170.699,32.471,156.103
C07832=1051.324,26.155,423.918,170.700,32.473,156.103
C07833=1051.331,26.405,423.901,170.702,32.475,156.104
C07834=1051.337,26.655,423.886,170.704,32.477,156.104
C07835=1051.343,26.904,423.870,170.705,32.479,156.104
C07836=1051.350,27.153,423.854,170.707,32.481,156.105
C07837=1051.356,27.403,423.838,170.709,32.483,156.105
C07838=1051.362,27.652,423.822,170.711,32.485,156.105
C07839=1051.368,27.901,423.806,170.712,32.487,156.105
C07840=1051.374,28.151,423.791,170.714,32.489,156.106
C07841=1051.380,28.400,423.774,170.715,32.491,156.106
C07842=1051.387,28.650,423.758,170.716,32.493,156.106
C07843=1051.393,28.900,423.742,170.718,32.495,156.107
C07844=1051.400,29.185,423.724,170.720,32.497,156.107
C07845=1051.407,29.471,423.705,170.722,32.500,156.107
C07846=1051.414,29.757,423.687,170.724,32.502,156.108
C07847=1051.422,30.043,423.668,170.726,32.505,156.108
C07848=1051.428,30.292,423.652,170.727,32.507,156.108
C07849=1051.434,30.542,423.636,170.729,32.509,156.109
C07850=1051.440,30.791,423.619,170.731,32.511,156.109
C07851=1051.445,31.041,423.603,170.732,32.513,156.109
C07852=1051.453,31.290,423.587,170.734,32.515,156.110
C07853=1051.459,31.540,423.571,170.736,32.517,156.110
C07854=1051.465,31.789,423.555,170.738,32.519,156.110
C07855=1051.471,32.038,423.538,170.739,32.521,156.111
C07856=1051.477,32.288,423.522,170.741,32.523,156.111
C07857=1051.483,32.537,423.506,170.743,32.525,156.111
C07858=1051.489,32.786,423.490,170.744,32.527,156.111
C07859=1051.496,33.036,423.474,170.746,32.529,156.112
C07860=1051.502,33.285,423.457,170.748,32.531,156.112
C07861=1051.508,33.535,423.441,170.749,32.533,156.112
C07862=1051.514,33.784,423.425,170.750,32.535,156.113
C07863=1051.520,34.033,423.409,170.752,32.537,156.113
C07864=1051.527,34.283,423.392,170.753,32.539,156.113
C07865=1051.533,34.533,423.376,170.755,32.541,156.114
C07866=1051.539,34.782,423.360,170.757,32.543,156.114
C07867=1051.545,35.031,423.344,170.758,32.545,156.114
C07868=1051.551,35.280,423.328,170.760,32.547,156.114
C07869=1051.558,35.530,423.311,170.762,32.549,156.115
C07870=1051.564,35.779,423.294,170.763,32.551,156.115
C07871=1051.570,36.028,423.278,170.765,32.553,156.115
C07872=1051.576,36.278,423.262,170.767,32.555,156.116
C07873=1051.583,36.528,423.245,170.769,32.557,156.116
C07874=1051.589,36.777,423.230,170.770,32.559,156.116
C07875=1051.595,37.026,423.213,170.772,32.561,156.117
C07876=1051.601,37.276,423.197,170.774,32.563,156.117
C07877=1051.608,37.525,423.180,170.775,32.565,156.117
C07878=1051.614,37.774,423.164,170.777,32.567,156.118
C07879=1051.620,38.024,423.147,170.779,32.569,156.118
C07880=1051.626,38.273,423.131,170.780,32.572,156.118
C07881=1051.633,38.523,423.114,170.782,32.574,156.119
C07882=1051.639,38.772,423.097,170.784,32.576,156.119
C07883=1051.645,39.021,423.081,170.785,32.578,156.119
C07884=1051.651,39.270,423.065,170.786,32.580,156.120
C07885=1051.657,39.521,423.048,170.788,32.582,156.120
C07886=1051.663,39.769,423.031,170.789,32.584,156.120
C07887=1051.669,40.019,423.015,170.791,32.586,156.120
C07888=1051.675,40.268,422.999,170.793,32.588,156.121
C07889=1051.682,40.517,422.981,170.794,32.591,156.121
C07890=1051.688,40.767,422.965,170.796,32.593,156.121
C07891=1051.693,41.016,422.948,170.798,32.595,156.122
C07892=1051.699,41.266,422.932,170.799,32.597,156.122
C07893=1051.706,41.515,422.915,170.801,32.599,156.122
C07894=1051.712,41.765,422.899,170.803,32.601,156.123
C07895=1051.718,42.014,422.882,170.804,32.603,156.123
C07896=1051.725,42.263,422.865,170.806,32.605,156.123
C07897=1051.731,42.513,422.849,170.808,32.607,156.124
C07898=1051.737,42.762,422.832,170.809,32.609,156.124
C07899=1051.743,43.011,422.815,170.811,32.611,156.124
C07900=1051.750,43.261,422.799,170.813,32.613,156.125
C07901=1051.756,43.510,422.782,170.814,32.615,156.125
C07902=1051.762,43.759,422.766,170.816,32.617,156.125
C07903=1051.768,44.009,422.748,170.817,32.619,156.126
C07904=1051.774,44.258,422.731,170.819,32.622,156.126
C07905=1051.780,44.507,422.715,170.821,32.624,156.126
C07906=1051.785,44.756,422.698,170.822,32.626,156.127
C07907=1051.792,45.006,422.681,170.824,32.628,156.127
C07908=1051.799,45.292,422.661,170.825,32.631,156.127
C07909=1051.806,45.578,422.643,170.827,32.633,156.128
C07910=1051.813,45.864,422.623,170.829,32.635,156.128
C07911=1051.819,46.150,422.604,170.831,32.638,156.128
C07912=1051.826,46.399,422.587,170.832,32.640,156.129
C07913=1051.832,46.648,422.570,170.834,32.643,156.129
C07914=1051.838,46.898,422.552,170.836,32.645,156.130
C07915=1051.844,47.148,422.536,170.837,32.647,156.130
C07916=1051.850,47.396,422.519,170.839,32.649,156.130
C07917=1051.856,47.647,422.502,170.840,32.651,156.130
C07918=1051.862,47.895,422.485,170.842,32.653,156.131
C07919=1051.868,48.144,422.468,170.844,32.655,156.131
C07920=1051.875,48.394,422.451,170.845,32.657,156.131
C07921=1051.880,48.643,422.434,170.847,32.659,156.132
C07922=1051.886,48.893,422.418,170.849,32.661,156.132
C07923=1051.893,49.142,422.400,170.850,32.664,156.133
C07924=1051.898,49.392,422.383,170.852,32.666,156.133
C07925=1051.905,49.641,422.366,170.854,32.668,156.133
C07926=1051.911,49.890,422.349,170.855,32.670,156.133
C07927=1051.917,50.139,422.332,170.857,32.673,156.134
C07928=1051.924,50.389,422.315,170.859,32.675,156.134
C07929=1051.929,50.638,422.299,170.860,32.677,156.134
C07930=1051.936,50.888,422.281,170.862,32.679,156.135
C07931=1051.942,51.137,422.264,170.863,32.680,156.135
C07932=1051.947,51.386,422.247,170.865,32.683,156.136
C07933=1051.954,51.636,422.229,170.867,32.685,156.136
C07934=1051.960,51.884,422.213,170.867,32.687,156.136
C07935=1051.966,52.135,422.195,170.869,32.689,156.136
C07936=1051.972,52.384,422.178,170.871,32.691,156.137
C07937=1051.978,52.632,422.161,170.872,32.694,156.137
C07938=1051.984,52.883,422.144,170.874,32.696,156.138
C07939=1051.991,53.131,422.127,170.876,32.698,156.138
C07940=1051.997,53.381,422.110,170.877,32.700,156.138
C07941=1052.003,53.630,422.092,170.879,32.702,156.138
C07942=1052.009,53.880,422.076,170.881,32.704,156.139
C07943=1052.015,54.129,422.058,170.882,32.706,156.139
C07944=1052.022,54.378,422.041,170.884,32.708,156.139
C07945=1052.028,54.627,422.024,170.885,32.710,156.140
C07946=1052.033,54.877,422.007,170.887,32.712,156.140
C07947=1052.040,55.126,421.990,170.889,32.714,156.140
C07948=1052.046,55.375,421.973,170.890,32.717,156.141
C07949=1052.053,55.625,421.955,170.892,32.719,156.141
C07950=1052.059,55.874,421.938,170.894,32.721,156.141
C07951=1052.065,56.124,421.920,170.895,32.723,156.142
C07952=1052.071,56.372,421.904,170.897,32.725,156.142
C07953=1052.078,56.622,421.886,170.899,32.727,156.142
C07954=1052.083,56.871,421.869,170.900,32.730,156.143
C07955=1052.090,57.121,421.852,170.902,32.732,156.143
C07956=1052.095,57.370,421.834,170.904,32.734,156.143
C07957=1052.102,57.619,421.817,170.905,32.736,156.144
C07958=1052.108,57.868,421.800,170.907,32.738,156.144
C07959=1052.115,58.118,421.782,170.909,32.740,156.144
C07960=1052.121,58.367,421.765,170.910,32.742,156.145
C07961=1052.127,58.617,421.748,170.912,32.744,156.145
C07962=1052.134,58.866,421.731,170.913,32.746,156.145
C07963=1052.140,59.115,421.714,170.915,32.748,156.146
C07964=1052.146,59.365,421.696,170.916,32.750,156.146
C07965=1052.152,59.614,421.679,170.917,32.752,156.146
C07966=1052.158,59.863,421.661,170.919,32.755,156.147
C07967=1052.165,60.112,421.644,170.921,32.757,156.147
C07968=1052.171,60.362,421.627,170.922,32.759,156.147
C07969=1052.178,60.611,421.609,170.924,32.761,156.148
C07970=1052.184,60.860,421.592,170.926,32.763,156.148
C07971=1052.190,61.110,421.574,170.927,32.765,156.148
C07972=1052.197,61.396,421.554,170.929,32.767,156.149
C07973=1052.205,61.681,421.534,170.931,32.770,156.149
C07974=1052.212,61.967,421.514,170.933,32.772,156.149
C07975=1052.219,62.253,421.494,170.935,32.775,156.150
C07976=1052.225,62.501,421.477,170.937,32.777,156.150
C07977=1052.231,62.751,421.459,170.938,32.779,156.151
C07978=1052.237,63.000,421.442,170.940,32.781,156.151
C07979=1052.244,63.249,421.425,170.942,32.783,156.151
C07980=1052.250,63.499,421.407,170.943,32.785,156.151
C07981=1052.257,63.748,421.390,170.945,32.787,156.152
C07982=1052.263,63.997,421.372,170.946,32.789,156.152
C07983=1052.270,64.247,421.354,170.948,32.791,156.152
C07984=1052.275,64.496,421.337,170.950,32.793,156.153
C07985=1052.281,64.746,421.319,170.951,32.795,156.153
C07986=1052.288,64.994,421.302,170.953,32.798,156.154
C07987=1052.294,65.244,421.284,170.955,32.800,156.154
C07988=1052.300,65.494,421.266,170.956,32.802,156.154
C07989=1052.305,65.743,421.248,170.958,32.804,156.154
C07990=1052.312,65.992,421.231,170.960,32.806,156.155
C07991=1052.318,66.241,421.213,170.961,32.808,156.155
C07992=1052.324,66.490,421.195,170.963,32.810,156.156
C07993=1052.331,66.740,421.178,170.964,32.812,156.156
C07994=1052.336,66.989,421.160,170.966,32.815,156.156
C07995=1052.343,67.239,421.142,170.968,32.817,156.157
C07996=1052.349,67.488,421.125,170.969,32.819,156.157
C07997=1052.355,67.737,421.107,170.971,32.821,156.157
C07998=1052.361,67.986,421.089,170.972,32.824,156.158
C07999=1052.367,68.235,421.071,170.973,32.825,156.158
C08000=1052.374,68.485,421.054,170.975,32.827,156.158
C08001=1052.380,68.734,421.036,170.977,32.830,156.159
C08002=1052.386,68.983,421.017,170.978,32.832,156.159
C08003=1052.392,69.233,420.999,170.980,32.834,156.159
C08004=1052.399,69.482,420.982,170.981,32.836,156.160
C08005=1052.404,69.731,420.965,170.983,32.839,156.160
C08006=1052.410,69.981,420.947,170.985,32.841,156.160
C08007=1052.417,70.230,420.928,170.986,32.843,156.161
C08008=1052.422,70.479,420.910,170.988,32.845,156.161
C08009=1052.428,70.729,420.892,170.990,32.847,156.161
C08010=1052.435,70.978,420.874,170.991,32.849,156.162
C08011=1052.441,71.227,420.857,170.993,32.851,156.162
C08012=1052.447,71.476,420.839,170.995,32.854,156.162
C08013=1052.454,71.725,420.820,170.996,32.856,156.163
C08014=1052.459,71.974,420.803,170.998,32.858,156.163
C08015=1052.465,72.224,420.785,170.999,32.860,156.164
C08016=1052.472,72.473,420.766,171.001,32.862,156.164
C08017=1052.477,72.722,420.749,171.003,32.864,156.164
C08018=1052.483,72.972,420.731,171.004,32.867,156.165
C08019=1052.490,73.221,420.712,171.006,32.869,156.165
C08020=1052.496,73.471,420.694,171.008,32.871,156.165
C08021=1052.502,73.720,420.677,171.009,32.873,156.166
C08022=1052.509,73.969,420.658,171.011,32.875,156.166
C08023=1052.515,74.219,420.640,171.012,32.877,156.166
C08024=1052.521,74.467,420.622,171.014,32.879,156.167
C08025=1052.527,74.717,420.604,171.016,32.882,156.167
C08026=1052.533,74.967,420.586,171.017,32.884,156.167
C08027=1052.539,75.216,420.568,171.019,32.886,156.168
C08028=1052.545,75.465,420.550,171.021,32.889,156.168
C08029=1052.551,75.714,420.531,171.022,32.891,156.168
C08030=1052.557,75.964,420.514,171.024,32.893,156.169
C08031=1052.564,76.213,420.495,171.026,32.895,156.169
C08032=1052.569,76.462,420.477,171.027,32.897,156.169
C08033=1052.576,76.711,420.459,171.029,32.899,156.170
C08034=1052.582,76.961,420.441,171.031,32.901,156.170
C08035=1052.588,77.210,420.422,171.032,32.904,156.170
C08036=1052.595,77.495,420.401,171.034,32.906,156.171
C08037=1052.603,77.780,420.381,171.036,32.908,156.171
C08038=1052.609,78.067,420.360,171.038,32.911,156.172
C08039=1052.616,78.352,420.340,171.040,32.914,156.172
C08040=1052.623,78.601,420.321,171.041,32.915,156.172
C08041=1052.628,78.849,420.303,171.043,32.918,156.173
C08042=1052.635,79.099,420.285,171.045,32.920,156.173
C08043=1052.640,79.349,420.265,171.046,32.922,156.173
C08044=1052.646,79.598,420.248,171.047,32.925,156.174
C08045=1052.652,79.847,420.229,171.048,32.927,156.174
C08046=1052.659,80.096,420.211,171.050,32.929,156.175
C08047=1052.665,80.346,420.193,171.052,32.931,156.175
C08048=1052.670,80.595,420.173,171.053,32.933,156.175
C08049=1052.677,80.845,420.155,171.055,32.936,156.176
C08050=1052.682,81.093,420.137,171.057,32.938,156.176
C08051=1052.689,81.342,420.119,171.058,32.940,156.176
C08052=1052.695,81.592,420.101,171.060,32.942,156.177
C08053=1052.701,81.841,420.082,171.061,32.944,156.177
C08054=1052.706,82.090,420.063,171.063,32.947,156.177
C08055=1052.713,82.340,420.045,171.065,32.949,156.178
C08056=1052.719,82.589,420.027,171.066,32.951,156.178
C08057=1052.725,82.838,420.008,171.068,32.953,156.179
C08058=1052.732,83.087,419.989,171.070,32.955,156.179
C08059=1052.737,83.337,419.971,171.071,32.957,156.179
C08060=1052.743,83.585,419.952,171.073,32.960,156.180
C08061=1052.749,83.835,419.934,171.075,32.962,156.180
C08062=1052.756,84.084,419.916,171.076,32.964,156.180
C08063=1052.762,84.333,419.897,171.078,32.966,156.181
C08064=1052.768,84.583,419.878,171.079,32.968,156.181
C08065=1052.774,84.832,419.859,171.081,32.971,156.181
C08066=1052.780,85.081,419.842,171.083,32.973,156.182
C08067=1052.786,85.330,419.823,171.084,32.975,156.182
C08068=1052.792,85.580,419.804,171.086,32.978,156.182
C08069=1052.798,85.829,419.785,171.088,32.980,156.183
C08070=1052.805,86.078,419.767,171.089,32.982,156.183
C08071=1052.811,86.328,419.749,171.091,32.984,156.184
C08072=1052.817,86.577,419.730,171.093,32.986,156.184
C08073=1052.823,86.826,419.711,171.094,32.988,156.184
C08074=1052.829,87.075,419.692,171.096,32.991,156.185
C08075=1052.835,87.324,419.674,171.098,32.993,156.185
C08076=1052.842,87.573,419.655,171.099,32.995,156.185
C08077=1052.847,87.823,419.637,171.101,32.997,156.186
C08078=1052.853,88.072,419.618,171.103,32.999,156.186
C08079=1052.860,88.321,419.599,171.104,33.001,156.186
C08080=1052.866,88.570,419.581,171.106,33.004,156.187
C08081=1052.872,88.820,419.561,171.107,33.006,156.187
C08082=1052.878,89.069,419.543,171.109,33.008,156.187
C08083=1052.885,89.318,419.524,171.111,33.010,156.188
C08084=1052.891,89.567,419.505,171.112,33.012,156.188
C08085=1052.897,89.817,419.487,171.114,33.014,156.188
C08086=1052.903,90.066,419.468,171.116,33.016,156.189
C08087=1052.909,90.315,419.450,171.117,33.019,156.189
C08088=1052.916,90.564,419.431,171.119,33.021,156.189
C08089=1052.921,90.813,419.412,171.121,33.023,156.190
C08090=1052.927,91.062,419.393,171.122,33.025,156.190
C08091=1052.933,91.312,419.374,171.124,33.027,156.191
C08092=1052.939,91.561,419.356,171.126,33.030,156.191
C08093=1052.945,91.810,419.336,171.127,33.032,156.191
C08094=1052.952,92.059,419.318,171.129,33.034,156.192
C08095=1052.957,92.309,419.298,171.131,33.036,156.192
C08096=1052.964,92.558,419.280,171.132,33.039,156.192
C08097=1052.969,92.807,419.261,171.134,33.041,156.193
C08098=1052.976,93.057,419.242,171.136,33.044,156.193
C08099=1052.981,93.306,419.223,171.137,33.045,156.194
C08100=1052.988,93.591,419.201,171.139,33.048,156.194
C08101=1052.995,93.876,419.179,171.141,33.051,156.194
C08102=1053.002,94.162,419.157,171.143,33.053,156.195
C08103=1053.009,94.447,419.135,171.145,33.056,156.195
C08104=1053.016,94.696,419.116,171.146,33.058,156.196
C08105=1053.021,94.946,419.097,171.148,33.060,156.196
C08106=1053.028,95.195,419.079,171.150,33.062,156.196
C08107=1053.033,95.444,419.059,171.151,33.064,156.197
C08108=1053.040,95.693,419.041,171.153,33.067,156.197
C08109=1053.046,95.942,419.021,171.155,33.069,156.197
C08110=1053.052,96.191,419.002,171.156,33.072,156.198
C08111=1053.058,96.441,418.983,171.158,33.074,156.198
C08112=1053.064,96.690,418.964,171.160,33.076,156.198
C08113=1053.070,96.939,418.945,171.161,33.078,156.199
C08114=1053.076,97.189,418.926,171.163,33.080,156.199
C08115=1053.082,97.437,418.906,171.165,33.083,156.200
C08116=1053.088,97.687,418.887,171.166,33.085,156.200
C08117=1053.095,97.936,418.868,171.168,33.087,156.200
C08118=1053.100,98.185,418.849,171.170,33.089,156.201
C08119=1053.107,98.434,418.831,171.171,33.091,156.201
C08120=1053.113,98.683,418.811,171.173,33.093,156.201
C08121=1053.119,98.932,418.792,171.175,33.096,156.202
C08122=1053.125,99.182,418.773,171.176,33.098,156.202
C08123=1053.130,99.431,418.753,171.178,33.100,156.203
C08124=1053.137,99.680,418.734,171.180,33.102,156.203
C08125=1053.143,99.929,418.715,171.181,33.104,156.203
C08126=1053.149,100.178,418.696,171.183,33.107,156.204
C08127=1053.156,100.428,418.677,171.185,33.109,156.204
C08128=1053.162,100.677,418.657,171.186,33.111,156.204
C08129=1053.168,100.926,418.638,171.188,33.113,156.205
C08130=1053.174,101.176,418.619,171.190,33.115,156.205
C08131=1053.180,101.425,418.599,171.191,33.118,156.205
C08132=1053.186,101.674,418.580,171.193,33.120,156.206
C08133=1053.192,101.923,418.561,171.195,33.122,156.206
C08134=1053.198,102.172,418.541,171.196,33.124,156.206
C08135=1053.203,102.421,418.522,171.198,33.127,156.207
C08136=1053.209,102.670,418.502,171.200,33.129,156.207
C08137=1053.216,102.919,418.483,171.201,33.131,156.208
C08138=1053.222,103.169,418.464,171.203,33.133,156.208
C08139=1053.228,103.418,418.444,171.205,33.136,156.208
C08140=1053.233,103.667,418.425,171.206,33.138,156.209
C08141=1053.239,103.916,418.405,171.208,33.140,156.209
C08142=1053.246,104.166,418.386,171.210,33.142,156.209
C08143=1053.252,104.415,418.366,171.211,33.145,156.210
C08144=1053.258,104.664,418.346,171.213,33.147,156.210
C08145=1053.264,104.913,418.327,171.215,33.150,156.211
C08146=1053.270,105.162,418.307,171.216,33.152,156.211
C08147=1053.275,105.412,418.288,171.218,33.154,156.211
C08148=1053.282,105.660,418.269,171.220,33.156,156.212
C08149=1053.288,105.910,418.249,171.221,33.159,156.212
C08150=1053.294,106.158,418.229,171.223,33.161,156.212
C08151=1053.300,106.408,418.210,171.225,33.163,156.213
C08152=1053.306,106.657,418.190,171.226,33.165,156.213
C08153=1053.312,106.906,418.171,171.228,33.167,156.214
C08154=1053.318,107.155,418.151,171.230,33.170,156.214
C08155=1053.324,107.405,418.132,171.231,33.172,156.214
C08156=1053.330,107.653,418.112,171.233,33.174,156.215
C08157=1053.336,107.903,418.093,171.235,33.176,156.215
C08158=1053.342,108.152,418.072,171.237,33.179,156.215
C08159=1053.348,108.401,418.053,171.238,33.181,156.216
C08160=1053.355,108.650,418.034,171.240,33.183,156.216
C08161=1053.361,108.899,418.014,171.242,33.185,156.217
C08162=1053.367,109.149,417.995,171.243,33.187,156.217
C08163=1053.373,109.398,417.974,171.245,33.190,156.217
C08164=1053.380,109.683,417.952,171.247,33.192,156.218
C08165=1053.387,109.969,417.929,171.249,33.195,156.218
C08166=1053.393,110.254,417.907,171.251,33.198,156.219
C08167=1053.401,110.539,417.884,171.253,33.200,156.219
C08168=1053.407,110.789,417.865,171.254,33.202,156.219
C08169=1053.413,111.037,417.845,171.256,33.204,156.220
C08170=1053.420,111.287,417.825,171.258,33.207,156.220
C08171=1053.425,111.536,417.806,171.260,33.209,156.220
C08172=1053.431,111.785,417.786,171.261,33.211,156.221
C08173=1053.437,112.034,417.766,171.263,33.213,156.221
C08174=1053.443,112.284,417.746,171.265,33.216,156.222
C08175=1053.449,112.533,417.726,171.266,33.218,156.222
C08176=1053.455,112.782,417.706,171.268,33.220,156.222
C08177=1053.461,113.031,417.686,171.270,33.222,156.223
C08178=1053.467,113.280,417.667,171.271,33.225,156.223
C08179=1053.474,113.530,417.647,171.273,33.227,156.223
C08180=1053.480,113.778,417.627,171.275,33.229,156.224
C08181=1053.486,114.027,417.607,171.277,33.231,156.224
C08182=1053.491,114.277,417.587,171.278,33.234,156.225
C08183=1053.497,114.526,417.567,171.280,33.236,156.225
C08184=1053.503,114.775,417.547,171.282,33.238,156.225
C08185=1053.509,115.024,417.527,171.283,33.241,156.226
C08186=1053.515,115.273,417.507,171.285,33.243,156.226
C08187=1053.521,115.522,417.486,171.287,33.246,156.227
C08188=1053.527,115.771,417.466,171.288,33.248,156.227
C08189=1053.533,116.021,417.447,171.290,33.250,156.227
C08190=1053.539,116.270,417.427,171.292,33.253,156.228
C08191=1053.544,116.519,417.406,171.293,33.255,156.228
C08192=1053.550,116.768,417.386,171.295,33.257,156.229
C08193=1053.557,117.017,417.366,171.297,33.260,156.229
C08194=1053.563,117.266,417.346,171.299,33.262,156.229
C08195=1053.568,117.515,417.325,171.300,33.264,156.230
C08196=1053.574,117.764,417.305,171.302,33.266,156.230
C08197=1053.580,118.013,417.285,171.304,33.269,156.230
C08198=1053.586,118.263,417.264,171.305,33.271,156.231
C08199=1053.592,118.511,417.244,171.307,33.273,156.231
C08200=1053.598,118.760,417.224,171.309,33.276,156.232
C08201=1053.604,119.010,417.205,171.311,33.278,156.232
C08202=1053.609,119.259,417.184,171.312,33.280,156.232
C08203=1053.615,119.508,417.164,171.314,33.282,156.233
C08204=1053.622,119.758,417.144,171.316,33.285,156.233
C08205=1053.628,120.007,417.124,171.317,33.287,156.234
C08206=1053.633,120.256,417.104,171.319,33.289,156.234
C08207=1053.639,120.505,417.084,171.321,33.292,156.234
C08208=1053.646,120.754,417.063,171.323,33.294,156.235
C08209=1053.651,121.003,417.042,171.324,33.296,156.235
C08210=1053.657,121.251,417.022,171.326,33.298,156.235
C08211=1053.664,121.501,417.002,171.328,33.301,156.236
C08212=1053.669,121.750,416.981,171.329,33.303,156.236
C08213=1053.675,121.999,416.961,171.331,33.306,156.237
C08214=1053.682,122.248,416.941,171.333,33.308,156.237
C08215=1053.688,122.497,416.921,171.335,33.310,156.237
C08216=1053.693,122.746,416.900,171.336,33.313,156.238
C08217=1053.700,122.996,416.880,171.338,33.315,156.238
C08218=1053.706,123.245,416.860,171.340,33.317,156.239
C08219=1053.711,123.494,416.839,171.342,33.319,156.239
C08220=1053.717,123.743,416.819,171.343,33.322,156.239
C08221=1053.724,123.991,416.798,171.345,33.324,156.240
C08222=1053.730,124.241,416.778,171.347,33.326,156.240
C08223=1053.736,124.490,416.758,171.349,33.328,156.240
C08224=1053.742,124.739,416.738,171.350,33.331,156.241
C08225=1053.747,124.989,416.717,171.352,33.333,156.241
C08226=1053.753,125.238,416.697,171.354,33.335,156.242
C08227=1053.760,125.486,416.676,171.356,33.338,156.242
C08228=1053.766,125.772,416.653,171.358,33.340,156.243
C08229=1053.773,126.057,416.630,171.360,33.343,156.243
C08230=1053.780,126.343,416.606,171.362,33.346,156.243
C08231=1053.787,126.628,416.582,171.364,33.348,156.244
C08232=1053.793,126.877,416.562,171.365,33.350,156.244
C08233=1053.799,127.127,416.541,171.367,33.353,156.245
C08234=1053.806,127.375,416.521,171.369,33.355,156.245
C08235=1053.812,127.624,416.500,171.371,33.357,156.245
C08236=1053.817,127.873,416.480,171.372,33.359,156.246
C08237=1053.824,128.122,416.459,171.374,33.362,156.246
C08238=1053.830,128.371,416.439,171.376,33.364,156.246
C08239=1053.836,128.621,416.418,171.378,33.366,156.247
C08240=1053.842,128.870,416.398,171.379,33.368,156.247
C08241=1053.849,129.119,416.377,171.381,33.371,156.248
C08242=1053.854,129.368,416.356,171.383,33.373,156.248
C08243=1053.861,129.617,416.336,171.385,33.375,156.248
C08244=1053.867,129.865,416.315,171.388,33.378,156.249
C08245=1053.873,130.115,416.294,171.389,33.380,156.249
C08246=1053.879,130.364,416.274,171.391,33.382,156.250
C08247=1053.885,130.613,416.253,171.393,33.384,156.250
C08248=1053.891,130.862,416.233,171.395,33.387,156.250
C08249=1053.898,131.112,416.213,171.396,33.389,156.251
C08250=1053.903,131.360,416.191,171.398,33.391,156.251
C08251=1053.910,131.610,416.171,171.400,33.393,156.251
C08252=1053.916,131.858,416.150,171.402,33.396,156.252
C08253=1053.922,132.108,416.129,171.404,33.398,156.252
C08254=1053.928,132.356,416.108,171.405,33.400,156.253
C08255=1053.934,132.606,416.087,171.407,33.403,156.253
C08256=1053.940,132.855,416.067,171.409,33.405,156.253
C08257=1053.945,133.103,416.046,171.411,33.408,156.254
C08258=1053.951,133.353,416.025,171.412,33.410,156.254
C08259=1053.957,133.601,416.004,171.414,33.412,156.255
C08260=1053.963,133.851,415.983,171.416,33.415,156.255
C08261=1053.969,134.100,415.962,171.418,33.417,156.255
C08262=1053.975,134.349,415.942,171.420,33.419,156.256
C08263=1053.981,134.598,415.921,171.421,33.422,156.256
C08264=1053.987,134.847,415.899,171.423,33.424,156.257
C08265=1053.994,135.096,415.879,171.425,33.426,156.257
C08266=1053.999,135.345,415.857,171.427,33.429,156.257
C08267=1054.005,135.595,415.836,171.429,33.431,156.258
C08268=1054.011,135.843,415.816,171.430,33.433,156.258
C08269=1054.017,136.093,415.795,171.432,33.436,156.259
C08270=1054.023,136.341,415.774,171.434,33.438,156.259
C08271=1054.030,136.590,415.752,171.436,33.440,156.259
C08272=1054.035,136.839,415.732,171.437,33.442,156.260
C08273=1054.041,137.088,415.710,171.439,33.445,156.260
C08274=1054.047,137.337,415.690,171.441,33.447,156.261
C08275=1054.053,137.586,415.669,171.443,33.449,156.261
C08276=1054.059,137.836,415.647,171.445,33.452,156.261
C08277=1054.065,138.085,415.626,171.447,33.454,156.262
C08278=1054.071,138.334,415.605,171.448,33.456,156.262
C08279=1054.077,138.582,415.584,171.450,33.459,156.263
C08280=1054.083,138.832,415.563,171.452,33.461,156.263
C08281=1054.089,139.081,415.542,171.454,33.463,156.263
C08282=1054.095,139.329,415.521,171.456,33.466,156.264
C08283=1054.101,139.579,415.500,171.457,33.468,156.264
C08284=1054.107,139.828,415.479,171.459,33.470,156.264
C08285=1054.113,140.077,415.457,171.461,33.473,156.265
C08286=1054.119,140.326,415.435,171.463,33.476,156.265
C08287=1054.125,140.575,415.416,171.465,33.478,156.266
C08288=1054.131,140.824,415.394,171.467,33.480,156.266
C08289=1054.137,141.073,415.373,171.469,33.483,156.267
C08290=1054.143,141.322,415.351,171.471,33.485,156.267
C08291=1054.149,141.570,415.330,171.473,33.487,156.267
C08292=1054.155,141.856,415.305,171.475,33.490,156.268
C08293=1054.162,142.141,415.281,171.477,33.493,156.268
C08294=1054.168,142.427,415.257,171.479,33.495,156.269
C08295=1054.176,142.711,415.232,171.481,33.498,156.269
C08296=1054.182,142.961,415.211,171.483,33.501,156.270
C08297=1054.188,143.210,415.189,171.485,33.503,156.270
C08298=1054.194,143.458,415.168,171.487,33.505,156.270
C08299=1054.200,143.707,415.146,171.489,33.508,156.271
C08300=1054.206,143.957,415.125,171.490,33.510,156.271
C08301=1054.211,144.206,415.104,171.492,33.512,156.272
C08302=1054.217,144.455,415.082,171.494,33.515,156.272
C08303=1054.224,144.704,415.061,171.496,33.517,156.272
C08304=1054.229,144.953,415.040,171.498,33.520,156.273
C08305=1054.236,145.202,415.019,171.500,33.522,156.273
C08306=1054.242,145.451,414.997,171.501,33.524,156.274
C08307=1054.248,145.699,414.976,171.503,33.527,156.274
C08308=1054.254,145.949,414.954,171.505,33.529,156.274
C08309=1054.260,146.198,414.932,171.507,33.531,156.275
C08310=1054.266,146.447,414.911,171.509,33.534,156.275
C08311=1054.272,146.695,414.889,171.511,33.536,156.276
C08312=1054.278,146.945,414.868,171.513,33.538,156.276
C08313=1054.284,147.194,414.846,171.514,33.541,156.277
C08314=1054.290,147.442,414.825,171.516,33.543,156.277
C08315=1054.296,147.692,414.803,171.518,33.546,156.277
C08316=1054.302,147.941,414.782,171.520,33.548,156.278
C08317=1054.308,148.190,414.760,171.522,33.551,156.278
C08318=1054.314,148.438,414.739,171.524,33.553,156.279
C08319=1054.320,148.688,414.717,171.526,33.555,156.279
C08320=1054.325,148.937,414.695,171.528,33.558,156.279
C08321=1054.331,149.186,414.674,171.530,33.560,156.280
C08322=1054.337,149.435,414.652,171.532,33.563,156.280
C08323=1054.343,149.684,414.630,171.534,33.565,156.281
C08324=1054.349,149.933,414.609,171.536,33.567,156.281
C08325=1054.355,150.181,414.587,171.538,33.570,156.281
C08326=1054.361,150.430,414.565,171.540,33.572,156.282
C08327=1054.368,150.680,414.543,171.541,33.574,156.282
C08328=1054.373,150.929,414.521,171.543,33.577,156.283
C08329=1054.379,151.178,414.500,171.545,33.579,156.283
C08330=1054.385,151.427,414.478,171.547,33.582,156.284
C08331=1054.391,151.675,414.456,171.549,33.585,156.284
C08332=1054.397,151.925,414.434,171.551,33.586,156.284
C08333=1054.402,152.173,414.412,171.553,33.589,156.285
C08334=1054.408,152.423,414.391,171.555,33.592,156.285
C08335=1054.414,152.672,414.369,171.556,33.594,156.286
C08336=1054.421,152.920,414.347,171.558,33.597,156.286
C08337=1054.427,153.169,414.326,171.560,33.599,156.286
C08338=1054.432,153.418,414.303,171.562,33.601,156.287
C08339=1054.438,153.668,414.282,171.564,33.604,156.287
C08340=1054.445,153.916,414.259,171.566,33.606,156.288
C08341=1054.451,154.165,414.238,171.568,33.609,156.288
C08342=1054.456,154.414,414.216,171.570,33.611,156.289
C08343=1054.462,154.663,414.194,171.572,33.613,156.289
C08344=1054.468,154.912,414.172,171.574,33.616,156.289
C08345=1054.474,155.161,414.150,171.575,33.618,156.290
C08346=1054.480,155.410,414.127,171.578,33.621,156.290
C08347=1054.486,155.659,414.106,171.580,33.623,156.291
C08348=1054.492,155.908,414.084,171.582,33.625,156.291
C08349=1054.498,156.157,414.061,171.584,33.628,156.291
C08350=1054.504,156.406,414.040,171.586,33.631,156.292
C08351=1054.510,156.655,414.018,171.588,33.633,156.292
C08352=1054.516,156.904,413.995,171.590,33.636,156.293
C08353=1054.522,157.153,413.974,171.592,33.638,156.293
C08354=1054.528,157.401,413.952,171.594,33.640,156.294
C08355=1054.533,157.651,413.929,171.596,33.643,156.294
C08356=1054.540,157.935,413.904,171.598,33.646,156.295
C08357=1054.546,158.220,413.879,171.600,33.648,156.295
C08358=1054.554,158.506,413.853,171.602,33.652,156.296
C08359=1054.561,158.790,413.828,171.604,33.654,156.296
C08360=1054.567,159.040,413.806,171.606,33.657,156.296
C08361=1054.573,159.288,413.784,171.608,33.659,156.297
C08362=1054.578,159.537,413.762,171.610,33.661,156.297
C08363=1054.584,159.786,413.740,171.612,33.664,156.298
C08364=1054.591,160.035,413.718,171.614,33.666,156.298
C08365=1054.596,160.284,413.695,171.616,33.669,156.299
C08366=1054.603,160.533,413.673,171.618,33.671,156.299
C08367=1054.608,160.782,413.650,171.620,33.674,156.299
C08368=1054.615,161.030,413.628,171.622,33.676,156.300
C08369=1054.620,161.280,413.606,171.625,33.679,156.300
C08370=1054.626,161.529,413.583,171.627,33.682,156.301
C08371=1054.631,161.777,413.562,171.628,33.684,156.301
C08372=1054.637,162.026,413.539,171.630,33.687,156.302
C08373=1054.643,162.275,413.516,171.632,33.689,156.302
C08374=1054.648,162.525,413.493,171.634,33.692,156.303
C08375=1054.655,162.773,413.471,171.636,33.694,156.303
C08376=1054.661,163.022,413.448,171.638,33.697,156.303
C08377=1054.666,163.272,413.426,171.640,33.699,156.304
C08378=1054.671,163.520,413.403,171.642,33.702,156.304
C08379=1054.678,163.768,413.381,171.644,33.704,156.305
C08380=1054.683,164.017,413.358,171.646,33.707,156.305
C08381=1054.689,164.267,413.336,171.648,33.710,156.306
C08382=1054.694,164.516,413.313,171.650,33.712,156.306
C08383=1054.701,164.764,413.291,171.652,33.715,156.307
C08384=1054.707,165.013,413.268,171.654,33.717,156.307
C08385=1054.712,165.263,413.245,171.656,33.720,156.308
C08386=1054.718,165.512,413.222,171.658,33.723,156.308
C08387=1054.724,165.760,413.200,171.660,33.725,156.308
C08388=1054.730,166.009,413.177,171.662,33.728,156.309
C08389=1054.735,166.257,413.155,171.664,33.730,156.309
C08390=1054.741,166.507,413.132,171.666,33.733,156.310
C08391=1054.747,166.755,413.110,171.668,33.735,156.310
C08392=1054.753,167.004,413.087,171.670,33.738,156.311
C08393=1054.758,167.253,413.064,171.672,33.741,156.311
C08394=1054.764,167.502,413.041,171.674,33.743,156.312
C08395=1054.770,167.751,413.018,171.676,33.746,156.312
C08396=1054.776,168.000,412.997,171.678,33.748,156.312
C08397=1054.782,168.249,412.974,171.680,33.751,156.313
C08398=1054.788,168.498,412.951,171.682,33.753,156.313
C08399=1054.793,168.747,412.928,171.684,33.756,156.314
C08400=1054.799,168.996,412.905,171.686,33.758,156.314
C08401=1054.806,169.244,412.882,171.688,33.761,156.315
C08402=1054.811,169.493,412.859,171.690,33.763,156.315
C08403=1054.817,169.742,412.836,171.692,33.766,156.316
C08404=1054.823,169.991,412.814,171.694,33.769,156.316
C08405=1054.828,170.240,412.791,171.696,33.771,156.316
C08406=1054.835,170.489,412.768,171.699,33.774,156.317
C08407=1054.841,170.737,412.745,171.701,33.777,156.317
C08408=1054.846,170.986,412.722,171.703,33.779,156.318
C08409=1054.853,171.236,412.699,171.705,33.782,156.318
C08410=1054.858,171.485,412.676,171.707,33.784,156.319
C08411=1054.865,171.733,412.654,171.709,33.787,156.319
C08412=1054.871,171.982,412.631,171.711,33.789,156.320
C08413=1054.876,172.231,412.608,171.713,33.792,156.320
C08414=1054.882,172.480,412.585,171.715,33.795,156.321
C08415=1054.888,172.729,412.562,171.717,33.797,156.321
C08416=1054.894,172.978,412.539,171.719,33.800,156.321
C08417=1054.900,173.226,412.517,171.721,33.802,156.322
C08418=1054.906,173.475,412.494,171.723,33.805,156.322
C08419=1054.911,173.724,412.471,171.725,33.807,156.323
C08420=1054.919,174.009,412.444,171.728,33.810,156.323
C08421=1054.925,174.294,412.418,171.730,33.813,156.324
C08422=1054.932,174.578,412.392,171.732,33.816,156.324
C08423=1054.939,174.862,412.365,171.736,33.819,156.325
C08424=1054.944,175.111,412.342,171.738,33.822,156.325
C08425=1054.951,175.360,412.320,171.740,33.824,156.326
C08426=1054.957,175.609,412.297,171.742,33.827,156.326
C08427=1054.963,175.858,412.273,171.744,33.829,156.327
C08428=1054.969,176.106,412.250,171.746,33.832,156.327
C08429=1054.975,176.355,412.227,171.748,33.834,156.328
C08430=1054.981,176.604,412.204,171.750,33.837,156.328
C08431=1054.986,176.853,412.181,171.752,33.840,156.328
C08432=1054.994,177.102,412.158,171.754,33.842,156.329
C08433=1054.999,177.351,412.135,171.756,33.845,156.329
C08434=1055.005,177.600,412.112,171.758,33.847,156.330
C08435=1055.011,177.848,412.089,171.760,33.850,156.330
C08436=1055.017,178.097,412.065,171.762,33.853,156.331
C08437=1055.023,178.346,412.042,171.765,33.855,156.331
C08438=1055.029,178.595,412.019,171.768,33.858,156.332
C08439=1055.035,178.844,411.996,171.770,33.860,156.332
C08440=1055.042,179.123,411.970,171.772,33.863,156.333
C08441=1055.049,179.401,411.944,171.774,33.866,156.333
C08442=1055.055,179.680,411.918,171.777,33.869,156.334
C08443=1055.062,179.958,411.892,171.779,33.872,156.334
C08444=1055.068,180.207,411.869,171.781,33.874,156.335
C08445=1055.074,180.455,411.845,171.783,33.877,156.335
C08446=1055.080,180.704,411.822,171.785,33.879,156.336
C08447=1055.086,180.953,411.799,171.787,33.882,156.336
C08448=1055.093,181.202,411.775,171.790,33.885,156.336
C08449=1055.098,181.451,411.752,171.792,33.887,156.337
C08450=1055.104,181.699,411.729,171.794,33.890,156.337
C08451=1055.111,181.949,411.706,171.796,33.893,156.338
C08452=1055.117,182.197,411.682,171.798,33.895,156.338
C08453=1055.123,182.446,411.659,171.801,33.898,156.339
C08454=1055.130,182.695,411.635,171.803,33.900,156.339
C08455=1055.136,182.944,411.612,171.805,33.903,156.340
C08456=1055.141,183.193,411.589,171.808,33.905,156.340
C08457=1055.148,183.442,411.565,171.810,33.908,156.341
C08458=1055.154,183.691,411.542,171.812,33.911,156.341
C08459=1055.160,183.939,411.519,171.814,33.913,156.341
C08460=1055.166,184.188,411.495,171.816,33.916,156.342
C08461=1055.172,184.437,411.472,171.818,33.919,156.342
C08462=1055.177,184.685,411.447,171.820,33.921,156.343
C08463=1055.184,184.935,411.424,171.822,33.924,156.343
C08464=1055.190,185.183,411.401,171.824,33.927,156.344
C08465=1055.195,185.432,411.377,171.827,33.929,156.344
C08466=1055.201,185.681,411.353,171.830,33.933,156.345
C08467=1055.207,185.930,411.329,171.832,33.935,156.345
C08468=1055.212,186.179,411.306,171.834,33.938,156.346
C08469=1055.218,186.427,411.281,171.836,33.941,156.346
C08470=1055.224,186.676,411.258,171.838,33.943,156.347
C08471=1055.230,186.925,411.234,171.840,33.946,156.347
C08472=1055.235,187.174,411.210,171.842,33.949,156.348
C08473=1055.241,187.422,411.187,171.845,33.951,156.348
C08474=1055.247,187.671,411.162,171.847,33.955,156.349
C08475=1055.253,187.920,411.139,171.849,33.957,156.349
C08476=1055.258,188.169,411.115,171.851,33.960,156.350
C08477=1055.265,188.418,411.091,171.853,33.963,156.350
C08478=1055.270,188.667,411.066,171.855,33.965,156.351
C08479=1055.276,188.915,411.043,171.858,33.968,156.351
C08480=1055.282,189.165,411.019,171.860,33.971,156.352
C08481=1055.288,189.413,410.995,171.863,33.973,156.352
C08482=1055.294,189.661,410.972,171.865,33.977,156.353
C08483=1055.300,189.911,410.947,171.867,33.979,156.353
C08484=1055.306,190.164,410.923,171.869,33.982,156.354
C08485=1055.311,190.419,410.898,171.871,33.985,156.354
C08486=1055.318,190.674,410.874,171.874,33.988,156.355
C08487=1055.323,190.928,410.849,171.876,33.990,156.355
C08488=1055.330,191.177,410.825,171.878,33.994,156.356
C08489=1055.335,191.425,410.801,171.880,33.996,156.356
C08490=1055.341,191.674,410.777,171.883,33.999,156.357
C08491=1055.347,191.923,410.753,171.885,34.002,156.357
C08492=1055.353,192.172,410.730,171.888,34.004,156.358
C08493=1055.359,192.421,410.705,171.890,34.007,156.358
C08494=1055.365,192.669,410.681,171.892,34.010,156.359
C08495=1055.371,192.919,410.657,171.894,34.013,156.359
C08496=1055.377,193.167,410.633,171.896,34.016,156.360
C08497=1055.382,193.415,410.609,171.899,34.019,156.360
C08498=1055.389,193.664,410.585,171.901,34.021,156.361
C08499=1055.394,193.913,410.560,171.903,34.024,156.361
C08500=1055.401,194.162,410.536,171.905,34.027,156.362
C08501=1055.406,194.411,410.512,171.907,34.029,156.362
C08502=1055.413,194.660,410.488,171.911,34.033,156.363
C08503=1055.418,194.908,410.464,171.913,34.035,156.363
C08504=1055.425,195.157,410.440,171.915,34.038,156.364
C08505=1055.430,195.406,410.416,171.917,34.041,156.364
C08506=1055.437,195.655,410.392,171.919,34.044,156.365
C08507=1055.442,195.903,410.367,171.922,34.046,156.365
C08508=1055.449,196.152,410.343,171.924,34.049,156.366
C08509=1055.454,196.400,410.318,171.926,34.052,156.366
C08510=1055.460,196.650,410.294,171.928,34.054,156.367
C08511=1055.466,196.898,410.270,171.931,34.058,156.367
C08512=1055.472,197.147,410.245,171.933,34.060,156.368
C08513=1055.478,197.395,410.222,171.936,34.063,156.368
C08514=1055.484,197.645,410.197,171.938,34.066,156.369
C08515=1055.491,197.893,410.172,171.941,34.069,156.369
C08516=1055.496,198.142,410.148,171.943,34.071,156.370
C08517=1055.503,198.391,410.124,171.945,34.075,156.370
C08518=1055.508,198.639,410.100,171.947,34.077,156.371
C08519=1055.514,198.888,410.075,171.950,34.080,156.371
C08520=1055.521,199.137,410.050,171.952,34.083,156.372
C08521=1055.526,199.385,410.026,171.954,34.086,156.372
C08522=1055.533,199.634,410.002,171.956,34.088,156.373
C08523=1055.538,199.883,409.978,171.960,34.092,156.373
C08524=1055.545,200.131,409.953,171.962,34.094,156.374
C08525=1055.551,200.381,409.929,171.964,34.097,156.375
C08526=1055.556,200.629,409.904,171.966,34.100,156.375
C08527=1055.563,200.878,409.880,171.969,34.103,156.376
C08528=1055.569,201.127,409.855,171.971,34.105,156.376
C08529=1055.575,201.375,409.831,171.973,34.108,156.377
C08530=1055.581,201.624,409.807,171.975,34.111,156.377
C08531=1055.587,201.873,409.781,171.978,34.114,156.378
C08532=1055.593,202.121,409.758,171.980,34.117,156.378
C08533=1055.600,202.370,409.732,171.983,34.120,156.379
C08534=1055.605,202.619,409.708,171.986,34.123,156.379
C08535=1055.611,202.867,409.683,171.988,34.125,156.380
C08536=1055.617,203.117,409.658,171.990,34.128,156.380
C08537=1055.622,203.365,409.634,171.992,34.132,156.381
C08538=1055.628,203.614,409.609,171.995,34.135,156.381
C08539=1055.634,203.862,409.584,171.997,34.137,156.382
C08540=1055.641,204.111,409.560,171.999,34.140,156.382
C08541=1055.647,204.360,409.535,172.002,34.143,156.383
C08542=1055.652,204.608,409.510,172.004,34.146,156.383
C08543=1055.658,204.857,409.485,172.007,34.149,156.384
C08544=1055.664,205.106,409.460,172.009,34.152,156.385
C08545=1055.670,205.355,409.436,172.012,34.155,156.385
C08546=1055.676,205.603,409.410,172.014,34.158,156.386
C08547=1055.682,205.852,409.385,172.016,34.161,156.386
C08548=1055.707,206.903,409.281,172.219,34.252,156.400
C08549=1055.713,207.141,409.256,172.220,34.255,156.400
C08550=1055.719,207.381,409.231,172.222,34.259,156.401
C08551=1055.725,207.620,409.206,172.225,34.262,156.402
C08552=1055.732,207.859,409.181,172.226,34.266,156.402
C08553=1055.738,208.098,409.157,172.228,34.270,156.403
C08554=1055.744,208.337,409.131,172.230,34.273,156.404
C08555=1055.749,208.576,409.106,172.232,34.277,156.405
C08556=1055.755,208.815,409.082,172.233,34.281,156.405
C08557=1055.762,209.063,409.056,172.236,34.284,156.406
C08558=1055.768,209.313,409.030,172.238,34.288,156.407
C08559=1055.775,209.561,409.004,172.240,34.292,156.407
C08560=1055.780,209.810,408.978,172.241,34.296,156.408
C08561=1055.787,210.058,408.952,172.243,34.299,156.409
C08562=1055.793,210.306,408.927,172.245,34.303,156.410
C08563=1055.799,210.555,408.900,172.248,34.307,156.410
C08564=1055.806,210.803,408.874,172.250,34.311,156.411
C08565=1055.812,211.052,408.848,172.251,34.315,156.412
C08566=1055.818,211.300,408.822,172.253,34.318,156.412
C08567=1055.824,211.549,408.796,172.255,34.322,156.413
C08568=1055.831,211.798,408.770,172.257,34.326,156.414
C08569=1055.837,212.046,408.743,172.260,34.330,156.415
C08570=1055.843,212.295,408.718,172.261,34.333,156.415
C08571=1055.849,212.543,408.691,172.263,34.337,156.416
C08572=1055.856,212.793,408.666,172.265,34.341,156.417
C08573=1055.862,213.041,408.639,172.267,34.345,156.418
C08574=1055.868,213.289,408.613,172.270,34.348,156.418
C08575=1055.874,213.537,408.586,172.272,34.352,156.419
C08576=1055.880,213.786,408.561,172.273,34.356,156.420
C08577=1055.886,214.035,408.534,172.275,34.360,156.421
C08578=1055.893,214.283,408.508,172.277,34.364,156.421
C08579=1055.898,214.532,408.482,172.279,34.367,156.422
C08580=1055.905,214.780,408.456,172.282,34.371,156.423
C08581=1055.911,215.029,408.429,172.284,34.375,156.424
C08582=1055.918,215.277,408.403,172.285,34.379,156.424
C08583=1055.924,215.526,408.376,172.287,34.382,156.425
C08584=1055.930,215.775,408.350,172.289,34.386,156.426
C08585=1055.936,216.023,408.324,172.292,34.390,156.426
C08586=1055.943,216.271,408.298,172.294,34.394,156.427
C08587=1055.948,216.520,408.271,172.296,34.397,156.428
C08588=1055.956,216.769,408.245,172.297,34.401,156.429
C08589=1055.961,217.018,408.219,172.299,34.405,156.429
C08590=1055.967,217.266,408.192,172.302,34.408,156.430
C08591=1055.974,217.515,408.166,172.304,34.413,156.431
C08592=1055.980,217.763,408.139,172.306,34.416,156.432
C08593=1055.986,218.011,408.113,172.308,34.420,156.432
C08594=1055.993,218.260,408.086,172.310,34.423,156.433
C08595=1055.999,218.508,408.060,172.312,34.427,156.434
C08596=1056.005,218.757,408.033,172.314,34.431,156.434
C08597=1056.012,219.005,408.007,172.316,34.434,156.435
C08598=1056.018,219.254,407.980,172.318,34.438,156.436
C08599=1056.024,219.503,407.953,172.320,34.442,156.437
C08600=1056.030,219.751,407.928,172.322,34.446,156.437
C08601=1056.036,220.000,407.901,172.325,34.449,156.438
C08602=1056.043,220.249,407.875,172.327,34.453,156.439
C08603=1056.049,220.497,407.848,172.329,34.457,156.439
C08604=1056.056,220.746,407.822,172.331,34.460,156.440
C08605=1056.062,220.987,407.795,172.332,34.464,156.441
C08606=1056.068,221.229,407.769,172.335,34.468,156.442
C08607=1056.074,221.470,407.743,172.337,34.471,156.442
C08608=1056.080,221.712,407.717,172.339,34.475,156.443
C08609=1056.086,221.953,407.691,172.341,34.478,156.444
C08610=1056.092,222.195,407.666,172.343,34.482,156.444
C08611=1056.098,222.436,407.640,172.345,34.486,156.445
C08612=1056.103,222.678,407.613,172.347,34.489,156.446
C08613=1056.110,222.927,407.586,172.349,34.493,156.447
C08614=1056.116,223.175,407.560,172.351,34.497,156.447
C08615=1056.123,223.423,407.533,172.353,34.501,156.448
C08616=1056.129,223.672,407.506,172.356,34.504,156.449
C08617=1056.135,223.921,407.479,172.358,34.508,156.450
C08618=1056.141,224.169,407.452,172.360,34.512,156.450
C08619=1056.147,224.418,407.426,172.362,34.515,156.451
C08620=1056.154,224.666,407.399,172.364,34.519,156.452
C08621=1056.160,224.914,407.372,172.367,34.523,156.452
C08622=1056.166,225.163,407.345,172.369,34.526,156.453
C08623=1056.172,225.412,407.318,172.370,34.530,156.454
C08624=1056.179,225.660,407.291,172.372,34.534,156.455
C08625=1056.184,225.908,407.264,172.374,34.538,156.455
C08626=1056.192,226.157,407.237,172.377,34.541,156.456
C08627=1056.197,226.405,407.211,172.379,34.545,156.457
C08628=1056.204,226.654,407.183,172.381,34.548,156.457
C08629=1056.210,226.902,407.156,172.383,34.552,156.458
C08630=1056.216,227.151,407.129,172.385,34.556,156.459
C08631=1056.222,227.399,407.102,172.388,34.559,156.460
C08632=1056.229,227.648,407.075,172.390,34.563,156.460
C08633=1056.235,227.896,407.049,172.392,34.567,156.461
C08634=1056.242,228.145,407.021,172.394,34.570,156.462
C08635=1056.248,228.393,406.995,172.396,34.574,156.462
C08636=1056.254,228.641,406.967,172.399,34.578,156.463
C08637=1056.261,228.890,406.940,172.401,34.582,156.464
C08638=1056.266,229.139,406.913,172.403,34.585,156.465
C08639=1056.273,229.387,406.885,172.405,34.589,156.465
C08640=1056.279,229.636,406.859,172.407,34.593,156.466
C08641=1056.286,229.884,406.831,172.410,34.596,156.467
C08642=1056.291,230.132,406.804,172.412,34.600,156.467
C08643=1056.298,230.381,406.777,172.414,34.603,156.468
C08644=1056.304,230.629,406.750,172.416,34.607,156.469
C08645=1056.310,230.878,406.722,172.418,34.611,156.470
C08646=1056.317,231.127,406.695,172.421,34.614,156.470
C08647=1056.323,231.374,406.668,172.423,34.618,156.471
C08648=1056.329,231.624,406.640,172.425,34.622,156.472
C08649=1056.335,231.872,406.613,172.427,34.626,156.473
C08650=1056.341,232.120,406.585,172.430,34.629,156.473
C08651=1056.347,232.368,406.559,172.432,34.633,156.474
C08652=1056.354,232.617,406.531,172.434,34.637,156.475
C08653=1056.360,232.866,406.504,172.436,34.640,156.475
C08654=1056.366,233.114,406.477,172.438,34.644,156.476
C08655=1056.373,233.362,406.449,172.441,34.647,156.477
C08656=1056.378,233.611,406.422,172.443,34.651,156.478
C08657=1056.385,233.859,406.394,172.445,34.655,156.478
C08658=1056.391,234.108,406.366,172.447,34.659,156.479
C08659=1056.397,234.356,406.339,172.450,34.662,156.480
C08660=1056.403,234.605,406.311,172.452,34.666,156.481
C08661=1056.411,234.900,406.279,172.454,34.670,156.481
C08662=1056.418,235.197,406.246,172.457,34.674,156.482
C08663=1056.426,235.493,406.213,172.460,34.679,156.483
C08664=1056.433,235.789,406.180,172.463,34.683,156.484
C08665=1056.440,236.038,406.152,172.465,34.687,156.485
C08666=1056.445,236.286,406.125,172.467,34.691,156.485
C08667=1056.451,236.535,406.097,172.469,34.694,156.486
C08668=1056.458,236.783,406.069,172.472,34.698,156.487
C08669=1056.464,237.031,406.042,172.474,34.702,156.488
C08670=1056.471,237.279,406.014,172.476,34.705,156.488
C08671=1056.477,237.528,405.986,172.478,34.709,156.489
C08672=1056.482,237.776,405.959,172.481,34.712,156.490
C08673=1056.488,237.991,405.935,172.483,34.716,156.490
C08674=1056.494,238.204,405.911,172.485,34.719,156.491
C08675=1056.499,238.418,405.887,172.487,34.722,156.492
C08676=1056.504,238.631,405.863,172.488,34.725,156.492
C08677=1056.510,238.845,405.840,172.490,34.728,156.493
C08678=1056.516,239.059,405.815,172.493,34.732,156.494
C08679=1056.521,239.274,405.792,172.495,34.735,156.494
C08680=1056.526,239.487,405.768,172.496,34.738,156.495
C08681=1056.533,239.736,405.740,172.499,34.741,156.495
C08682=1056.539,239.983,405.713,172.502,34.745,156.496
C08683=1056.545,240.232,405.684,172.504,34.748,156.497
C08684=1056.551,240.481,405.656,172.506,34.752,156.498
C08685=1056.558,240.729,405.629,172.508,34.756,156.498
C08686=1056.563,240.977,405.601,172.510,34.759,156.499
C08687=1056.570,241.225,405.573,172.513,34.763,156.500
C08688=1056.577,241.474,405.545,172.515,34.766,156.500
C08689=1056.583,241.723,405.517,172.517,34.770,156.501
C08690=1056.589,241.971,405.489,172.520,34.774,156.502
C08691=1056.595,242.219,405.461,172.523,34.777,156.503
C08692=1056.601,242.468,405.434,172.525,34.781,156.503
C08693=1056.608,242.716,405.405,172.527,34.785,156.504
C08694=1056.614,242.964,405.377,172.529,34.789,156.505
C08695=1056.620,243.212,405.349,172.532,34.792,156.506
C08696=1056.626,243.461,405.321,172.534,34.796,156.506
C08697=1056.632,243.709,405.293,172.536,34.799,156.507
C08698=1056.638,243.958,405.264,172.538,34.803,156.508
C08699=1056.645,244.206,405.236,172.541,34.807,156.508
C08700=1056.651,244.454,405.208,172.544,34.810,156.509
C08701=1056.657,244.702,405.180,172.546,34.814,156.510
C08702=1056.663,244.951,405.152,172.548,34.818,156.511
C08703=1056.669,245.199,405.123,172.550,34.821,156.511
C08704=1056.676,245.448,405.095,172.553,34.825,156.512
C08705=1056.682,245.697,405.067,172.555,34.828,156.513
C08706=1056.688,245.944,405.040,172.558,34.832,156.513
C08707=1056.694,246.192,405.010,172.560,34.836,156.514
C08708=1056.700,246.441,404.982,172.563,34.840,156.515
C08709=1056.706,246.690,404.954,172.565,34.843,156.516
C08710=1056.713,246.938,404.925,172.567,34.847,156.516
C08711=1056.719,247.186,404.897,172.569,34.850,156.517
C08712=1056.725,247.434,404.868,172.572,34.854,156.518
C08713=1056.731,247.683,404.840,172.575,34.858,156.519
C08714=1056.737,247.931,404.812,172.577,34.862,156.519
C08715=1056.744,248.179,404.783,172.579,34.865,156.520
C08716=1056.750,248.428,404.755,172.582,34.869,156.521
C08717=1056.755,248.662,404.728,172.584,34.873,156.522
C08718=1056.761,248.897,404.701,172.586,34.876,156.522
C08719=1056.767,249.132,404.673,172.588,34.879,156.523
C08720=1056.772,249.367,404.647,172.591,34.883,156.524
C08721=1056.778,249.602,404.620,172.593,34.886,156.524
C08722=1056.784,249.836,404.593,172.595,34.890,156.525
C08723=1056.790,250.071,404.566,172.597,34.893,156.526
C08724=1056.796,250.305,404.539,172.599,34.897,156.526
C08725=1056.802,250.554,404.511,172.603,34.900,156.527
C08726=1056.808,250.802,404.482,172.605,34.904,156.528
C08727=1056.814,251.050,404.452,172.607,34.908,156.529
C08728=1056.821,251.299,404.425,172.610,34.912,156.529
C08729=1056.827,251.547,404.396,172.612,34.915,156.530
C08730=1056.833,251.795,404.368,172.615,34.919,156.531
C08731=1056.839,252.043,404.339,172.617,34.922,156.532
C08732=1056.845,252.291,404.310,172.620,34.926,156.532
C08733=1056.851,252.540,404.281,172.622,34.930,156.533
C08734=1056.857,252.788,404.252,172.625,34.933,156.534
C08735=1056.864,253.036,404.223,172.627,34.937,156.534
C08736=1056.870,253.284,404.196,172.630,34.940,156.535
C08737=1056.877,253.533,404.166,172.632,34.944,156.536
C08738=1056.883,253.781,404.137,172.634,34.948,156.537
C08739=1056.889,254.029,404.109,172.637,34.952,156.537
C08740=1056.895,254.278,404.080,172.640,34.955,156.538
C08741=1056.901,254.526,404.051,172.642,34.959,156.539
C08742=1056.907,254.774,404.022,172.644,34.962,156.540
C08743=1056.913,255.023,403.994,172.647,34.966,156.540
C08744=1056.920,255.271,403.965,172.650,34.970,156.541
C08745=1056.927,255.519,403.936,172.652,34.973,156.542
C08746=1056.933,255.767,403.907,172.654,34.977,156.542
C08747=1056.940,256.016,403.878,172.657,34.980,156.543
C08748=1056.946,256.264,403.849,172.660,34.984,156.544
C08749=1056.952,256.512,403.820,172.662,34.988,156.545
C08750=1056.958,256.761,403.791,172.664,34.991,156.545
C08751=1056.964,257.009,403.762,172.667,34.995,156.546
C08752=1056.971,257.257,403.733,172.670,34.998,156.547
C08753=1056.977,257.505,403.704,172.672,35.002,156.548
C08754=1056.983,257.753,403.675,172.675,35.006,156.548
C08755=1056.989,258.001,403.646,172.677,35.009,156.549
C08756=1056.996,258.249,403.617,172.680,35.013,156.550
C08757=1057.003,258.498,403.588,172.682,35.016,156.550
C08758=1057.010,258.746,403.559,172.685,35.020,156.551
C08759=1057.015,258.995,403.531,172.687,35.023,156.552
C08760=1057.022,259.243,403.502,172.690,35.027,156.553
C08761=1057.028,259.491,403.473,172.693,35.031,156.553
C08762=1057.034,259.739,403.444,172.695,35.034,156.554
C08763=1057.041,259.987,403.414,172.698,35.038,156.555
C08764=1057.048,260.235,403.385,172.701,35.041,156.555
C08765=1057.054,260.484,403.356,172.703,35.045,156.556
C08766=1057.060,260.732,403.327,172.705,35.049,156.557
C08767=1057.066,260.980,403.298,172.709,35.052,156.558
C08768=1057.073,261.228,403.268,172.711,35.056,156.558
C08769=1057.079,261.477,403.239,172.713,35.059,156.559
C08770=1057.086,261.725,403.210,172.716,35.063,156.560
C08771=1057.092,261.973,403.181,172.719,35.066,156.561
C08772=1057.098,262.221,403.152,172.721,35.070,156.561
C08773=1057.104,262.455,403.124,172.724,35.074,156.562
C08774=1057.111,262.689,403.097,172.726,35.077,156.563
C08775=1057.117,262.923,403.069,172.729,35.080,156.563
C08776=1057.123,263.156,403.041,172.731,35.084,156.564
C08777=1057.129,263.390,403.013,172.733,35.087,156.565
C08778=1057.134,263.624,402.986,172.736,35.090,156.565
C08779=1057.140,263.858,402.958,172.739,35.094,156.566
C08780=1057.146,264.091,402.930,172.741,35.097,156.567
C08781=1057.152,264.339,402.901,172.743,35.101,156.568
C08782=1057.159,264.587,402.871,172.747,35.105,156.568
C08783=1057.165,264.835,402.842,172.749,35.108,156.569
C08784=1057.171,265.084,402.812,172.751,35.112,156.570
C08785=1057.178,265.332,402.783,172.754,35.116,156.571
C08786=1057.184,265.580,402.753,172.757,35.119,156.571
C08787=1057.190,265.828,402.724,172.760,35.123,156.572
C08788=1057.197,266.076,402.694,172.762,35.127,156.573
C08789=1057.203,266.325,402.665,172.764,35.130,156.573
C08790=1057.209,266.572,402.634,172.768,35.134,156.574
C08791=1057.215,266.821,402.605,172.770,35.137,156.575
C08792=1057.222,267.069,402.576,172.772,35.142,156.576
C08793=1057.228,267.317,402.546,172.776,35.145,156.577
C08794=1057.234,267.565,402.517,172.778,35.149,156.577
C08795=1057.241,267.813,402.487,172.781,35.152,156.578
C08796=1057.247,268.062,402.457,172.783,35.156,156.579
C08797=1057.253,268.309,402.427,172.786,35.159,156.579
C08798=1057.259,268.558,402.397,172.789,35.163,156.580
C08799=1057.266,268.806,402.367,172.791,35.167,156.581
C08800=1057.272,269.054,402.337,172.795,35.171,156.582
C08801=1057.278,269.302,402.308,172.797,35.174,156.582
C08802=1057.285,269.550,402.278,172.799,35.178,156.583
C08803=1057.291,269.799,402.248,172.803,35.181,156.584
C08804=1057.297,270.046,402.218,172.805,35.185,156.585
C08805=1057.304,270.295,402.188,172.808,35.189,156.585
C08806=1057.310,270.543,402.159,172.810,35.193,156.586
C08807=1057.316,270.791,402.128,172.813,35.196,156.587
C08808=1057.323,271.039,402.098,172.816,35.200,156.588
C08809=1057.328,271.287,402.068,172.818,35.203,156.588
C08810=1057.335,271.535,402.039,172.822,35.207,156.589
C08811=1057.341,271.783,402.008,172.824,35.211,156.590
C08812=1057.348,272.032,401.979,172.827,35.215,156.591
C08813=1057.354,272.280,401.948,172.829,35.218,156.591
C08814=1057.360,272.528,401.918,172.832,35.222,156.592
C08815=1057.366,272.775,401.888,172.835,35.225,156.593
C08816=1057.372,273.025,401.858,172.837,35.229,156.594
C08817=1057.379,273.272,401.828,172.841,35.233,156.594
C08818=1057.385,273.520,401.798,172.843,35.237,156.595
C08819=1057.391,273.768,401.767,172.846,35.240,156.596
C08820=1057.398,274.016,401.738,172.849,35.244,156.597
C08821=1057.404,274.264,401.707,172.852,35.248,156.598
C08822=1057.410,274.512,401.676,172.854,35.251,156.598
C08823=1057.416,274.760,401.647,172.857,35.255,156.599
C08824=1057.423,275.009,401.617,172.860,35.259,156.600
C08825=1057.428,275.257,401.586,172.863,35.263,156.601
C08826=1057.436,275.505,401.556,172.865,35.266,156.601
C08827=1057.441,275.753,401.526,172.868,35.270,156.602
C08828=1057.448,276.001,401.495,172.871,35.273,156.603
C08829=1057.454,276.237,401.466,172.873,35.277,156.603
C08830=1057.460,276.472,401.438,172.877,35.280,156.604
C08831=1057.466,276.708,401.409,172.879,35.284,156.605
C08832=1057.472,276.943,401.380,172.881,35.288,156.606
C08833=1057.478,277.179,401.352,172.884,35.291,156.606
C08834=1057.484,277.415,401.322,172.887,35.295,156.607
C08835=1057.490,277.650,401.293,172.890,35.298,156.608
C08836=1057.496,277.886,401.264,172.892,35.302,156.609
C08837=1057.502,278.134,401.234,172.895,35.305,156.609
C08838=1057.509,278.382,401.204,172.898,35.309,156.610
C08839=1057.515,278.630,401.173,172.900,35.312,156.611
C08840=1057.521,278.878,401.142,172.904,35.317,156.612
C08841=1057.528,279.127,401.111,172.906,35.320,156.612
C08842=1057.534,279.374,401.081,172.909,35.324,156.613
C08843=1057.541,279.623,401.051,172.913,35.327,156.614
C08844=1057.547,279.870,401.021,172.915,35.331,156.615
C08845=1057.553,280.118,400.989,172.918,35.335,156.615
C08846=1057.559,280.366,400.959,172.920,35.338,156.616
C08847=1057.566,280.615,400.928,172.924,35.343,156.617
C08848=1057.571,280.863,400.898,172.926,35.346,156.618
C08849=1057.578,281.110,400.866,172.929,35.350,156.619
C08850=1057.584,281.358,400.836,172.932,35.354,156.619
C08851=1057.590,281.607,400.805,172.935,35.357,156.620
C08852=1057.596,281.854,400.774,172.937,35.361,156.621
C08853=1057.603,282.103,400.744,172.941,35.365,156.622
C08854=1057.609,282.351,400.713,172.943,35.369,156.622
C08855=1057.615,282.598,400.682,172.946,35.373,156.623
C08856=1057.622,282.847,400.651,172.950,35.376,156.624
C08857=1057.628,283.094,400.620,172.952,35.380,156.625
C08858=1057.634,283.342,400.589,172.955,35.384,156.626
C08859=1057.641,283.591,400.559,172.958,35.387,156.626
C08860=1057.647,283.838,400.527,172.961,35.391,156.627
C08861=1057.653,284.087,400.497,172.963,35.395,156.628
C08862=1057.659,284.334,400.466,172.967,35.399,156.629
C08863=1057.666,284.582,400.435,172.970,35.403,156.630
C08864=1057.673,284.830,400.404,172.972,35.406,156.630
C08865=1057.678,285.078,400.373,172.976,35.410,156.631
C08866=1057.685,285.326,400.342,172.978,35.414,156.632
C08867=1057.692,285.575,400.311,172.981,35.418,156.633
C08868=1057.698,285.822,400.280,172.985,35.421,156.633
C08869=1057.704,286.070,400.249,172.987,35.425,156.634
C08870=1057.711,286.318,400.218,172.990,35.429,156.635
C08871=1057.717,286.565,400.187,172.993,35.432,156.636
C08872=1057.723,286.814,400.156,172.996,35.436,156.637
C08873=1057.730,287.062,400.125,172.999,35.440,156.637
C08874=1057.737,287.310,400.093,173.002,35.443,156.638
C08875=1057.742,287.558,400.062,173.005,35.448,156.639
C08876=1057.749,287.806,400.031,173.007,35.451,156.640
C08877=1057.755,288.054,399.999,173.011,35.455,156.640
C08878=1057.762,288.302,399.969,173.014,35.459,156.641
C08879=1057.768,288.549,399.938,173.016,35.462,156.642
C08880=1057.775,288.797,399.906,173.020,35.466,156.643
C08881=1057.781,289.045,399.875,173.023,35.470,156.644
C08882=1057.786,289.293,399.844,173.026,35.474,156.644
C08883=1057.793,289.541,399.812,173.029,35.478,156.645
C08884=1057.800,289.789,399.781,173.032,35.482,156.646
C08885=1057.805,290.030,399.751,173.035,35.485,156.647
C08886=1057.812,290.271,399.719,173.038,35.489,156.647
C08887=1057.818,290.512,399.690,173.040,35.493,156.648
C08888=1057.825,290.753,399.659,173.044,35.496,156.649
C08889=1057.831,290.995,399.628,173.046,35.500,156.650
C08890=1057.836,291.236,399.597,173.049,35.504,156.651
C08891=1057.843,291.477,399.567,173.053,35.508,156.651
C08892=1057.849,291.718,399.536,173.055,35.511,156.652
C08893=1057.855,291.966,399.504,173.058,35.515,156.653
C08894=1057.862,292.214,399.473,173.062,35.519,156.654
C08895=1057.869,292.462,399.441,173.064,35.523,156.655
C08896=1057.874,292.709,399.410,173.067,35.526,156.655
C08897=1057.881,292.957,399.378,173.071,35.531,156.656
C08898=1057.887,293.205,399.347,173.073,35.534,156.657
C08899=1057.893,293.453,399.315,173.076,35.538,156.658
C08900=1057.900,293.701,399.283,173.080,35.542,156.659
C08901=1057.907,293.949,399.252,173.082,35.546,156.659
C08902=1057.912,294.197,399.220,173.086,35.550,156.660
C08903=1057.919,294.445,399.189,173.089,35.553,156.661
C08904=1057.926,294.692,399.157,173.092,35.557,156.662
C08905=1057.932,294.941,399.125,173.095,35.561,156.663
C08906=1057.938,295.189,399.094,173.098,35.565,156.664
C08907=1057.945,295.436,399.061,173.101,35.569,156.664
C08908=1057.951,295.684,399.030,173.104,35.573,156.665
C08909=1057.957,295.932,398.998,173.107,35.577,156.666
C08910=1057.964,296.180,398.966,173.110,35.580,156.667
C08911=1057.970,296.427,398.934,173.114,35.584,156.668
C08912=1057.977,296.675,398.902,173.116,35.588,156.668
C08913=1057.983,296.923,398.870,173.120,35.592,156.669
C08914=1057.989,297.171,398.838,173.123,35.596,156.670
C08915=1057.996,297.419,398.806,173.125,35.600,156.671
C08916=1058.002,297.667,398.774,173.129,35.604,156.672
C08917=1058.008,297.915,398.742,173.132,35.608,156.673
C08918=1058.014,298.163,398.709,173.136,35.612,156.673
C08919=1058.020,298.410,398.678,173.138,35.616,156.674
C08920=1058.026,298.658,398.646,173.141,35.620,156.675
C08921=1058.032,298.906,398.614,173.145,35.624,156.676
C08922=1058.039,299.153,398.581,173.148,35.628,156.677
C08923=1058.045,299.401,398.549,173.150,35.632,156.678
C08924=1058.052,299.649,398.517,173.154,35.636,156.679
C08925=1058.058,299.897,398.485,173.157,35.639,156.679
C08926=1058.064,300.145,398.452,173.161,35.644,156.680
C08927=1058.070,300.393,398.420,173.163,35.648,156.681
C08928=1058.077,300.640,398.388,173.166,35.652,156.682
C08929=1058.083,300.888,398.356,173.170,35.656,156.683
C08930=1058.089,301.136,398.323,173.173,35.659,156.684
C08931=1058.095,301.384,398.291,173.177,35.663,156.684
C08932=1058.101,301.632,398.258,173.179,35.667,156.685
C08933=1058.108,301.879,398.226,173.182,35.672,156.686
C08934=1058.114,302.127,398.194,173.186,35.676,156.687
C08935=1058.121,302.375,398.161,173.189,35.679,156.688
C08936=1058.127,302.622,398.129,173.192,35.683,156.689
C08937=1058.133,302.871,398.097,173.195,35.687,156.689
C08938=1058.140,303.118,398.064,173.198,35.691,156.690
C08939=1058.146,303.366,398.032,173.202,35.695,156.691
C08940=1058.152,303.614,398.000,173.205,35.700,156.692
C08941=1058.159,303.864,397.966,173.209,35.703,156.693
C08942=1058.166,304.113,397.934,173.211,35.707,156.694
C08943=1058.171,304.363,397.901,173.214,35.711,156.695
C08944=1058.178,304.613,397.868,173.218,35.715,156.695
C08945=1058.184,304.861,397.835,173.221,35.719,156.696
C08946=1058.191,305.109,397.804,173.225,35.723,156.697
C08947=1058.198,305.357,397.771,173.228,35.727,156.698
C08948=1058.204,305.605,397.738,173.231,35.732,156.699
C08949=1058.210,305.852,397.705,173.234,35.735,156.700
C08950=1058.217,306.100,397.672,173.237,35.739,156.701
C08951=1058.223,306.347,397.640,173.241,35.743,156.701
C08952=1058.229,306.595,397.607,173.244,35.747,156.702
C08953=1058.237,306.843,397.574,173.247,35.751,156.703
C08954=1058.243,307.091,397.542,173.251,35.755,156.704
C08955=1058.249,307.339,397.510,173.254,35.759,156.705
C08956=1058.256,307.586,397.477,173.258,35.764,156.706
C08957=1058.262,307.834,397.444,173.260,35.767,156.707
C08958=1058.269,308.082,397.411,173.264,35.771,156.707
C08959=1058.275,308.330,397.378,173.267,35.775,156.708
C08960=1058.281,308.577,397.346,173.270,35.779,156.709
C08961=1058.288,308.825,397.313,173.274,35.783,156.710
C08962=1058.296,309.072,397.280,173.277,35.787,156.711
C08963=1058.302,309.320,397.247,173.281,35.791,156.712
C08964=1058.308,309.568,397.214,173.284,35.796,156.713
C08965=1058.314,309.815,397.181,173.288,35.800,156.714
C08966=1058.321,310.063,397.148,173.291,35.804,156.714
C08967=1058.328,310.311,397.115,173.294,35.808,156.715
C08968=1058.334,310.559,397.083,173.297,35.812,156.716
C08969=1058.341,310.807,397.050,173.300,35.816,156.717
C08970=1058.347,311.054,397.016,173.304,35.819,156.718
C08971=1058.354,311.301,396.983,173.307,35.823,156.719
C08972=1058.361,311.550,396.950,173.310,35.827,156.720
C08973=1058.367,311.797,396.918,173.314,35.832,156.720
C08974=1058.373,312.045,396.885,173.317,35.836,156.721
C08975=1058.381,312.292,396.852,173.321,35.840,156.722
C08976=1058.387,312.540,396.819,173.324,35.844,156.723
C08977=1058.394,312.788,396.786,173.328,35.848,156.724
C08978=1058.401,313.036,396.753,173.331,35.852,156.725
C08979=1058.407,313.283,396.720,173.335,35.856,156.726
C08980=1058.414,313.531,396.686,173.338,35.860,156.727
C08981=1058.420,313.778,396.652,173.341,35.864,156.728
C08982=1058.427,314.027,396.619,173.345,35.869,156.729
C08983=1058.432,314.275,396.586,173.348,35.873,156.729
C08984=1058.439,314.521,396.552,173.352,35.877,156.730
C08985=1058.445,314.769,396.520,173.355,35.881,156.731
C08986=1058.452,315.017,396.485,173.359,35.885,156.732
C08987=1058.458,315.264,396.452,173.362,35.889,156.733
C08988=1058.464,315.513,396.418,173.365,35.893,156.734
C08989=1058.471,315.760,396.385,173.368,35.898,156.735
C08990=1058.477,316.008,396.351,173.372,35.902,156.736
C08991=1058.484,316.255,396.318,173.375,35.906,156.737
C08992=1058.489,316.503,396.284,173.379,35.911,156.738
C08993=1058.496,316.750,396.251,173.382,35.915,156.739
C08994=1058.502,316.998,396.216,173.385,35.919,156.739
C08995=1058.509,317.246,396.184,173.389,35.923,156.740
C08996=1058.515,317.494,396.149,173.392,35.928,156.741
C08997=1058.521,317.748,396.115,173.396,35.932,156.742
C08998=1058.528,318.002,396.080,173.399,35.936,156.743
C08999=1058.535,318.255,396.046,173.404,35.941,156.744
C09000=1058.542,318.509,396.011,173.407,35.945,156.745
C09001=1058.548,318.757,395.977,173.411,35.949,156.746
C09002=1058.555,319.004,395.944,173.414,35.953,156.747
C09003=1058.561,319.252,395.910,173.418,35.958,156.748
C09004=1058.568,319.499,395.876,173.421,35.962,156.749
C09005=1058.574,319.747,395.842,173.425,35.966,156.750
C09006=1058.580,319.996,395.808,173.428,35.971,156.751
C09007=1058.587,320.243,395.774,173.432,35.975,156.752
C09008=1058.593,320.491,395.740,173.435,35.979,156.753
C09009=1058.600,320.738,395.707,173.439,35.983,156.754
C09010=1058.606,320.986,395.672,173.442,35.987,156.754
C09011=1058.613,321.233,395.639,173.446,35.992,156.755
C09012=1058.619,321.481,395.604,173.449,35.996,156.756
C09013=1058.626,321.728,395.571,173.453,36.001,156.757
C09014=1058.632,321.976,395.536,173.456,36.005,156.758
C09015=1058.639,322.224,395.502,173.460,36.009,156.759
C09016=1058.645,322.471,395.469,173.463,36.013,156.760
C09017=1058.652,322.719,395.434,173.467,36.018,156.761
C09018=1058.659,322.966,395.400,173.470,36.022,156.762
C09019=1058.665,323.214,395.366,173.475,36.027,156.763
C09020=1058.672,323.461,395.332,173.478,36.031,156.764
C09021=1058.679,323.709,395.298,173.482,36.035,156.765
C09022=1058.685,323.957,395.264,173.485,36.039,156.766
C09023=1058.692,324.204,395.230,173.489,36.044,156.767
C09024=1058.698,324.452,395.196,173.492,36.048,156.768
C09025=1058.705,324.699,395.162,173.496,36.052,156.769
C09026=1058.712,324.947,395.127,173.499,36.056,156.770
C09027=1058.718,325.194,395.093,173.503,36.061,156.771
C09028=1058.725,325.442,395.059,173.507,36.066,156.772
C09029=1058.731,325.689,395.025,173.511,36.070,156.773
C09030=1058.738,325.937,394.991,173.514,36.074,156.774
C09031=1058.745,326.184,394.956,173.518,36.078,156.775
C09032=1058.752,326.432,394.921,173.521,36.083,156.776
C09033=1058.759,326.680,394.888,173.525,36.087,156.777
C09034=1058.765,326.927,394.854,173.528,36.091,156.777
C09035=1058.771,327.175,394.818,173.533,36.096,156.778
C09036=1058.779,327.422,394.785,173.536,36.100,156.779
C09037=1058.785,327.670,394.750,173.540,36.105,156.780
C09038=1058.792,327.918,394.715,173.543,36.109,156.781
C09039=1058.799,328.166,394.681,173.547,36.113,156.782
C09040=1058.805,328.412,394.646,173.550,36.118,156.783
C09041=1058.812,328.660,394.612,173.555,36.122,156.784
C09042=1058.819,328.908,394.578,173.558,36.126,156.785
C09043=1058.826,329.155,394.543,173.562,36.131,156.786
C09044=1058.832,329.403,394.509,173.565,36.136,156.787
C09045=1058.840,329.650,394.474,173.569,36.140,156.788
C09046=1058.846,329.898,394.440,173.573,36.144,156.789
C09047=1058.853,330.146,394.405,173.577,36.149,156.790
C09048=1058.860,330.393,394.371,173.581,36.153,156.791
C09049=1058.867,330.641,394.336,173.584,36.158,156.792
C09050=1058.873,330.887,394.301,173.588,36.162,156.793
C09051=1058.879,331.135,394.266,173.592,36.166,156.794
C09052=1058.886,331.383,394.231,173.596,36.171,156.795
C09053=1058.892,331.632,394.196,173.599,36.176,156.796
C09054=1058.900,331.880,394.161,173.603,36.180,156.797
C09055=1058.906,332.128,394.125,173.606,36.185,156.798
C09056=1058.913,332.377,394.091,173.611,36.189,156.799
C09057=1058.919,332.624,394.055,173.615,36.194,156.800
C09058=1058.926,332.872,394.021,173.618,36.198,156.801
C09059=1058.933,333.119,393.986,173.622,36.203,156.802
C09060=1058.939,333.367,393.951,173.626,36.208,156.803
C09061=1058.946,333.614,393.916,173.630,36.212,156.804
C09062=1058.952,333.862,393.880,173.633,36.217,156.805
C09063=1058.959,334.110,393.845,173.637,36.222,156.807
C09064=1058.965,334.357,393.810,173.642,36.226,156.808
C09065=1058.972,334.605,393.775,173.645,36.231,156.809
C09066=1058.979,334.852,393.740,173.649,36.235,156.810
C09067=1058.986,335.099,393.705,173.652,36.240,156.811
C09068=1058.992,335.347,393.670,173.657,36.245,156.812
C09069=1058.999,335.594,393.635,173.660,36.249,156.813
C09070=1059.006,335.841,393.600,173.664,36.254,156.814
C09071=1059.013,336.089,393.564,173.669,36.258,156.815
C09072=1059.020,336.336,393.529,173.672,36.263,156.816
C09073=1059.026,336.583,393.494,173.676,36.268,156.817
C09074=1059.032,336.831,393.458,173.679,36.272,156.818
C09075=1059.039,337.079,393.423,173.684,36.277,156.819
C09076=1059.046,337.326,393.388,173.687,36.282,156.820
C09077=1059.053,337.574,393.351,173.691,36.287,156.821
C09078=1059.060,337.821,393.316,173.696,36.291,156.822
C09079=1059.066,338.068,393.281,173.699,36.296,156.823
C09080=1059.073,338.316,393.246,173.703,36.301,156.824
C09081=1059.079,338.563,393.210,173.708,36.305,156.825
C09082=1059.086,338.810,393.174,173.711,36.310,156.826
C09083=1059.093,339.058,393.139,173.715,36.315,156.828
C09084=1059.099,339.305,393.103,173.719,36.320,156.829
C09085=1059.106,339.552,393.068,173.723,36.325,156.830
C09086=1059.113,339.800,393.032,173.727,36.329,156.831
C09087=1059.119,340.048,392.996,173.731,36.334,156.832
C09088=1059.127,340.294,392.961,173.735,36.339,156.833
C09089=1059.133,340.542,392.925,173.738,36.343,156.834
C09090=1059.139,340.789,392.890,173.743,36.349,156.835
C09091=1059.147,341.037,392.853,173.747,36.353,156.836
C09092=1059.153,341.285,392.818,173.750,36.358,156.837
C09093=1059.160,341.531,392.782,173.755,36.363,156.838
C09094=1059.167,341.779,392.747,173.759,36.367,156.839
C09095=1059.173,342.026,392.710,173.763,36.372,156.841
C09096=1059.181,342.274,392.675,173.767,36.377,156.842
C09097=1059.188,342.521,392.639,173.770,36.382,156.843
C09098=1059.194,342.768,392.603,173.775,36.387,156.844
C09099=1059.201,343.016,392.567,173.779,36.392,156.845
C09100=1059.207,343.263,392.531,173.783,36.397,156.846
C09101=1059.215,343.510,392.495,173.787,36.401,156.847
C09102=1059.221,343.757,392.459,173.791,36.406,156.848
C09103=1059.228,344.005,392.423,173.795,36.411,156.849
C09104=1059.235,344.252,392.387,173.799,36.416,156.851
C09105=1059.242,344.499,392.351,173.804,36.421,156.852
C09106=1059.249,344.747,392.314,173.807,36.426,156.853
